FUNCTION "Line.FCMain" : VOID	// FC 50
VERSION : 0.1
VAR_TEMP
  Alarm_Emergency : BOOL ;
  Rich_manuale : BOOL ;
  Rich_automatico : BOOL ;
END_VAR
BEGIN
NETWORK
TITLE =
      CALL  "Line.FCMapE";
      CALL  "Line.FCConfig";
NETWORK
TITLE =
      CALL  "Bench.Alarms" (
           NumDBallarmi             := "Line.Alarms",
           Reset_Allarmi            := "Line.Systems".Command.Reset_allarmi,
           AllarmeEmergenza         := "Line".Diagnostic.Alarm_Emergency,
           AllarmeStopCiclo         := "Line".Diagnostic.Alarm_Stop_Cycle,
           AllarmeStartCiclo        := "Line".Diagnostic.Alarm_No_Restart,
           AllarmeWarning           := "Line".Diagnostic.Alarm_Warning);
// cumula gli stati di emergenza per evitare definizioni errate degli stati macchina!
      A     "Line".Diagnostic.Alarm_Emergency;
      O     "OP10".Diagnostic.Alarm_Emergency;
      O     "OP20".Diagnostic.Alarm_Emergency;
      O     "OP40".Diagnostic.Alarm_Emergency;
      =     #Alarm_Emergency;
      A     "Line.MapE".S_Manuale;
      =     #Rich_manuale;
      A     "Line.MapE".S_Automatico;
      A     "Line.Systems".State.Porte_chiuse;
      =     #Rich_automatico;
      CALL  "Bench.Mode" (
           Enable                   := TRUE,
           AllarmeEmergenza         := #Alarm_Emergency,
           AusiliariOK              := "Line.MapE".Aux_OK,
           ComandoTestMacchina      := FALSE,
           ComandoSetup             := FALSE,
           ComandoManuale           := #Rich_manuale,
           ComandoAutomatico        := #Rich_automatico,
           TimerTest                := T 1,
           ModoEmergenza            := "Line".Mode.Emergency,
           ModoTestMacchina         := "Line".Mode.Test_Machine,
           ModoSetup                := "Line".Mode.Setup,
           ModoManuale              := "Line".Mode.Manual,
           ModoAutomatico           := "Line".Mode.Automatic,
           DO_PlcOk                 := "Line.Systems".State.PLC_OK);
      A     "Line.MapE".S_Manuale;
      FP    "M100.3";
      =     "FP_manual";
      A     "Line.MapE".S_Automatico;
      FP    "M100.5";
      =     "Fp_Automatic";
      A     "FP_manual";
      O     "Fp_Automatic";
      ON    "Line.MapE".Aux_OK;
      R     "Line.OperatorPanel".States.Op10_recipe;
      R     "Line.OperatorPanel".States.Op20_recipe;
      R     "Line.OperatorPanel".States.Op40_recipe;
NETWORK
TITLE =
      CALL  "Line.FCSystems";
      CALL  "Line.FCOperatorPanel";
      CALL  "Line.FCCycles";
NETWORK
TITLE =
      CALL  "Line.FCMapA";
END_FUNCTION

FUNCTION "Line.FCMapE" : VOID	// FC 51
VERSION : 0.1
BEGIN
NETWORK
TITLE =
      A     I 0.0;
      =     "Line.MapE".Q_Ribaditrice;
      A     I 0.1;
      =     "Line.MapE".Q_protezione_uscite;
      A     I 0.2;
      =     "Line.MapE".Q_Protez_circ_emergena;
      A     I 0.3;
      =     "Line.MapE".Q_Automatici_230_V;
      A     I 0.4;
      =     "Line.MapE".Aux_OK;
      A     I 0.5;
      =     "Line.MapE".Ripari_OK;
      A     I 0.6;
      =     "Line.MapE".Anomalia_Condizionatore;
      A     I 0.7;
      =     "Line.MapE".Sequenza_fasi_OK;
NETWORK
TITLE =
      A     I 1.0;
      =     "Line.MapE".PLC_OK;
      A     I 1.1;
      =     "Line.MapE".Chiave_Blocc_Porta_SX;
      A     I 1.2;
      =     "Line.MapE".Chiave_Blocc_Porta_DX;
      A     I 1.3;
      =     "Line.MapE".P_TestLampade;
      A     I 1.4;
      =     "Line.MapE".P_StartCiclo;
      AN    I 1.5;
      =     "Line.MapE".P_StopCiclo;
      A     I 1.7;
      =     "Line.MapE".S_Manuale;
      A     I 1.6;
      =     "Line.MapE".S_Automatico;
NETWORK
TITLE =
      A     I 2.0;
      =     "Line.MapE".Q_Azionam_Asse_X;
      A     I 2.1;
      =     "Line.MapE".Q_Azionam_Asse_Y;
      A     I 6.2;
      =     "Line.MapE".Jog_piu;
      A     I 6.3;
      =     "Line.MapE".Jog_meno;
      A     I 6.4;
      =     "Line.MapE".P_reset_allarmi;
      A     I 6.5;
      =     "Line.MapE".Pressostato_aria;
      A     I 7.6;
      =     "Line.MapE".Ribaditrice_bassa;
      A     I 7.5;
      =     "Line.MapE".Ribaditrice_alta;
NETWORK
TITLE =
      A     I 6.6;
      =     "Line.MapE".Press_aria_dpoop_EMG;
      A     I 2.2;
      =     "Line.MapE".Extracorsa_X;
      A     I 4.7;
      =     "Line.MapE".Extracorsa_Y;
END_FUNCTION

FUNCTION "Line.FCMapA" : VOID	// FC 52
VERSION : 0.1
BEGIN
NETWORK
TITLE =
      A     "Line.MapA".PLC_OK;
      =     Q 0.0;
// tolto!
//      UN    "Line.MapA".Valvola_generale_aria
//      =     A      3.5
      A     "Line.MapA".Marcia_ribaditrice;
      =     Q 1.0;
      A     "Line.MapA".EV_abbassa_ribaditrice;
      =     Q 1.1;
//      U     "Line.MapA".Spare_0_4
//      =     A      1.2
      A     "Line.MapA".Blocco_porta_SX;
      =     Q 3.6;
      A     "Line.MapA".Blocco_porta_DX;
      =     Q 3.7;
      A     "Line.MapA".Lampeggiante_allarmi;
      =     Q 0.7;
      A     "Line.MapA".LampPorteChiuse;
      =     Q 1.7;
END_FUNCTION

FUNCTION "Line.FCConfig" : VOID	// FC 53
VERSION : 0.1
BEGIN
NETWORK
TITLE =
      L     L#100;
      T     "Line.Config".Accel_assi_auto;
      T     "Line.Config".Accel_assi_man;
// Impostate da pagina Config su OP
//      L     L#15000
//      T     "Line.Config".Vel_max_assi_auto
////      T     "Line.Config".Vel_max_assi_man
//      L     L#71501
//      T     "Line.Config".Offset_attrezzo_OP10_X
//      L     L#47116
//      T     "Line.Config".Offset_attrezzo_OP10_Y
//      L     L#371523
//      T     "Line.Config".Offset_attrezzo_OP40_X
//      L     L#47047
//      T     "Line.Config".Offset_attrezzo_OP40_Y
END_FUNCTION

FUNCTION "Line.FCSystems" : VOID	// FC 55
VERSION : 0.1
VAR_TEMP
  Cmd_Marcia_ribaditrice : BOOL ;
  Cmd_Marcia_ribaditr_ibl : BOOL ;
  Cmd_abbassa_rib : BOOL ;
  Cmd_alza_rib : BOOL ;
  Cmd_abbassa_rib_ibl : BOOL ;
  Cmd_alza_rib_ibl : BOOL ;
  StartPosizX : BOOL ;
  StartPosizX_ibl : BOOL ;
  JogPiuX : BOOL ;
  JogMenoX : BOOL ;
  JogPiuX_ibl : BOOL ;
  JogMenoX_ibl : BOOL ;
  StartPosizY : BOOL ;
  StartPosizY_ibl : BOOL ;
  JogPiuY : BOOL ;
  JogMenoY : BOOL ;
  JogPiuY_ibl : BOOL ;
  JogMenoY_ibl : BOOL ;
  Profi_w_error : BOOL ;
  Profi_r_error : BOOL ;
  Override : INT ;
  Velocita_asse_X : DINT ;
  Velocita_asse_Y : DINT ;
  TeachIn_page_OP10 : BOOL ;
  TeachIn_page_OP40 : BOOL ;
  Punt1 : DINT ;
  PuntoSelezionato : INT ;
  Pos_comandata_asse_X : DINT ;
  Pos_comandata_asse_Y : DINT ;
  Tempo_ribaditura : DINT ;
END_VAR
BEGIN
NETWORK
TITLE = ******************       Diagnostica       *******************
NETWORK
TITLE = Diagnostica: Reset Allarmi
      A     "Line.MapE".P_reset_allarmi;
      FP    "AppoFP_M50.0";
      O(;
      A     "Line.OperatorPanel".Commands.Reset_Allarmi;
      FP    "AppoFP_M50.1";
      );
      S     "Line.Systems".Command.Reset_allarmi;
      A     "Line.Systems".Command.Reset_allarmi;
      L     S5T#500MS;
      SD    "TempoResetAllarmi";
      A     "TempoResetAllarmi";
      R     "Line.Systems".Command.Reset_allarmi;
NETWORK
TITLE = Allarmi di emergenza
      AN    "Line.MapE".Q_protezione_uscite;
      O(;
      A     "Line.Alarms".Emegency.Alarm01;
      AN    "Line.Systems".Command.Reset_allarmi;
      );
      =     "Line.Alarms".Emegency.Alarm01;
      AN    "Line.MapE".Q_Protez_circ_emergena;
      O(;
      A     "Line.Alarms".Emegency.Alarm02;
      AN    "Line.Systems".Command.Reset_allarmi;
      );
      =     "Line.Alarms".Emegency.Alarm02;
      AN    "Line.MapE".Sequenza_fasi_OK;
      =     "Line.Alarms".Emegency.Alarm03;
      AN    "Line.MapE".Q_Azionam_Asse_X;
      O(;
      A     "Line.Alarms".Emegency.Alarm04;
      AN    "Line.Systems".Command.Reset_allarmi;
      );
      =     "Line.Alarms".Emegency.Alarm04;
      AN    "Line.MapE".Q_Azionam_Asse_Y;
      O(;
      A     "Line.Alarms".Emegency.Alarm05;
      AN    "Line.Systems".Command.Reset_allarmi;
      );
      =     "Line.Alarms".Emegency.Alarm05;
      A     "Line.MapA".PLC_OK;
      AN    "Line.MapE".PLC_OK;
      O(;
      AN    "Line.MapA".PLC_OK;
      A     "Line.MapE".PLC_OK;
      );
      L     S5T#500MS;
      SD    "T_All_Rientro_PLC_OK";
      A     "T_All_Rientro_PLC_OK";
      S     "Line.Alarms".Emegency.Alarm14;
NETWORK
TITLE = Extracorsa Assi: Allarmi Emergenza
NETWORK
TITLE = Allarmi di STOP CICLO
      AN    "Line.MapE".Aux_OK;
      =     "Line.Alarms".StopCycle.Alarm11;
NETWORK
TITLE = Allarmi di NON START CICLO
NETWORK
TITLE = Allarmi di Warning
      AN    "Line.MapE".Q_Ribaditrice;
//      O(    
//      U     DB54.DBX   24.0
//      UN    DB55.DBX    0.0
//      )     
      =     "Line.Alarms".Warning.Alarm01;
      AN    "Line.MapE".Q_Automatici_230_V;
      =     "Line.Alarms".Warning.Alarm02;
      A     "Line.MapE".Anomalia_Condizionatore;
      =     "Line.Alarms".Warning.Alarm03;
NETWORK
TITLE = Diagnostica: Hold Macchina
      AN    "Line".Diagnostic.Alarm_Emergency;
      A(;
      A     "Line".Mode.Automatic;
      AN    "Line".Diagnostic.Alarm_Stop_Cycle;
      A     "Line.Systems".State.Porte_chiuse_e_bloccate;
      O(;
      A     "Line".Mode.Manual;
      A     "Line.Systems".State.Porte_chiuse;
      );
      );
      =     "Line".Diagnostic.Safe_State;
NETWORK
TITLE = ******************          Stati            *******************
      A     "Op10.Bench.Systems".State.Cassetto_fuori;
      O     "Op10.Bench.Systems".State.Cassetto_dentro;
      A     "Op10.Bench.Systems".State.Index_cassetto_alto;
      =     "Line.Systems".State.Cassetto_OP10_indexato;
      A     "Op40.Bench.Systems".State.Cassetto_fuori;
      O     "Op40.Bench.Systems".State.Cassetto_dentro;
      A     "Op40.Bench.Systems".State.Index_cassetto_alto;
      =     "Line.Systems".State.Cassetto_OP40_indexato;
NETWORK
TITLE =
      A     "Line.MapE".Ripari_OK;
      =     "Line.Systems".State.Porte_chiuse;
NETWORK
TITLE = Stato: Fronte Start Ciclo
NETWORK
TITLE = Lampade
      AN    "Line.Systems".State.Porte_chiuse;
      A     "Clock-T=0,8 sec.";
      O     "Line.Systems".State.Porte_chiuse;
      =     "Line.MapA".LampPorteChiuse;
NETWORK
TITLE = Pagina attiva di TeachIn
// Trovo quale stazione è in pagina di gestione punti
      L     "Line.OperatorPanel".OP_System_Data.PageDisplayed;
      L     21;
      ==I;
      =     #TeachIn_page_OP10;
      L     "Line.OperatorPanel".OP_System_Data.PageDisplayed;
      L     31;
      ==I;
      =     #TeachIn_page_OP40;
NETWORK
TITLE = ******************         Sistemi           *******************
NETWORK
TITLE = Uscita PLC OK
      A     "Line.Systems".State.PLC_OK;
      =     "Line.MapA".PLC_OK;
NETWORK
TITLE = Valvola generale aria
//      UN    "Line".Mode.Emergency
//      =     "Line.MapA".Valvola_generale_aria
      A     "Line.MapE".Aux_OK;
      AN    "Line.MapE".Press_aria_dpoop_EMG;
      O(;
      AN    "Line.MapE".Aux_OK;
      A     "Line.MapE".Press_aria_dpoop_EMG;
      );
      L     S5T#3S;
      SD    "T_Allarme_aria_compressa";
      A     "T_Allarme_aria_compressa";
      A     "Line.MapE".Aux_OK;
      ON    "Line.MapE".Pressostato_aria;
      O(;
      A     "Line.Alarms".Emegency.Alarm06;
      AN    "Line.Systems".Command.Reset_allarmi;
      );
      =     "Line.Alarms".Emegency.Alarm06;
      A     "T_Allarme_aria_compressa";
      AN    "Line.MapE".Aux_OK;
      O(;
      A     "Line.Alarms".Emegency.Alarm07;
      AN    "Line.Systems".Command.Reset_allarmi;
      );
      =     "Line.Alarms".Emegency.Alarm07;
NETWORK
TITLE = Prenotazione ribaditrice
      A     "Op10.Bench.Systems".Command.Prenota_ribaditrice;
      =     "Line.Systems".Command.PrenotaRib_OP10;
      A     "Op40.Bench.Systems".Command.Prenota_ribaditrice;
      =     "Line.Systems".Command.PrenotaRib_OP40;
      A     "Line.Cycles".Coord_Ribaditrice.State.State_Bit[10];
      =     "Line.Systems".State.Ribad_prenotata_da_OP10;
      A     "Line.Cycles".Coord_Ribaditrice.State.State_Bit[20];
      =     "Line.Systems".State.Ribad_prenotata_da_OP40;
NETWORK
TITLE = Marcia ribaditrice
//*************************** COMANDI DA CICLI *************************
      A     "Op10.Bench.Systems".Command.Marcia_ribaditrice;
      A     "Line.Systems".Command.PrenotaRib_OP10;
      O(;
      A     "Op40.Bench.Systems".Command.Marcia_ribaditrice;
      A     "Line.Systems".Command.PrenotaRib_OP40;
      );
      =     "Line.Systems".Command.Marcia_ribaditrice;
//*************************** COMANDI SENZA INTERBLOCCHI ***************
// Autoritenuta comando di marcia manuale
      A     "Line.OperatorPanel".Commands.Man_Marcia_Ribaditrice;
      A     "Line.MapE".Jog_piu;
      O     "Line.Systems".State.Ribadit_Motore_in_marcia;
      A     "Line".Mode.Manual;
      A(;
      AN    "Line.MapE".Jog_meno;
      ON    "Line.OperatorPanel".Commands.Man_Marcia_Ribaditrice;
      );
      AN    "Line.Alarms".Warning.Alarm05;
      A(;
      L     "Line.OperatorPanel".OP_System_Data.PageDisplayed;
      L     20;
      ==I;
      O(;
      L     "Line.OperatorPanel".OP_System_Data.PageDisplayed;
      L     30;
      ==I;
      );
      );
      =     "Line.Systems".Command.Marcia_manuale_ribaditr;
//CMD---------->Comando Marcia ribaditrice
//MANUALE
      A     "Line.Systems".Command.Marcia_manuale_ribaditr;
      A     "Line".Mode.Manual;
//AUTOMATICO
      O(;
      A     "Line".Mode.Automatic;
      AN    "Line".Diagnostic.Hold_State;
      A     "Line.Systems".Command.Marcia_ribaditrice;
      );
//SICUREZZA
      A     "Line".Diagnostic.Safe_State;
      A     "Line.MapE".Q_Ribaditrice;
      =     #Cmd_Marcia_ribaditrice;
//************************** INTERBLOCCHI (E SEGNALAZIONE) ****************************
//MSG---> Segnalazione interblocco Movimento ribaditrice non ammesso con motore ribaditrice in marcia
//      U     "Line.Systems".Command.Reset_allarmi
//      O(    
//      U     "Line.Systems".State.Cassetto_OP10_indexato
//      U     "Line.Systems".State.Cassetto_OP40_indexato
//      )     
//      R     "Line.Alarms".Warning.Alarm05
//      U     #Cmd_Marcia_ribaditrice
//      U(    
//      UN    "Line.Systems".State.Cassetto_OP10_indexato
//      ON    "Line.Systems".State.Cassetto_OP40_indexato
//      )     
//      S     "Line.Alarms".Warning.Alarm05
//************************** COMANDI CON INTERBLOCCHI ******************************
//CMD-------------> Comando Marcia
      A     #Cmd_Marcia_ribaditrice;
      AN    "Line.Alarms".Warning.Alarm05;
      =     #Cmd_Marcia_ribaditr_ibl;
      =     "Line.Systems".State.Ribadit_Motore_in_marcia;
      =     "Line.MapA".Marcia_ribaditrice;
NETWORK
TITLE = Alza/abbassa ribaditrice
//*************************** COMANDI DA CICLI *************************
      A     "Op10.Bench.Systems".Command.Abbassa_ribaditrice;
      A     "Line.Systems".Command.PrenotaRib_OP10;
      O(;
      A     "Op40.Bench.Systems".Command.Abbassa_ribaditrice;
      A     "Line.Systems".Command.PrenotaRib_OP40;
      );
      =     "Line.Systems".Command.Abbassa_ribaditrice;
      A     "Op10.Bench.Systems".Command.Alza_ribaditrice;
      A     "Line.Systems".Command.PrenotaRib_OP10;
      O(;
      A     "Op40.Bench.Systems".Command.Alza_ribaditrice;
      A     "Line.Systems".Command.PrenotaRib_OP40;
      );
      =     "Line.Systems".Command.Alza_ribaditrice;
//*************************** COMANDI SENZA INTERBLOCCHI ***************
//CMD---------->Comando abbassa ribaditrice
//MANUALE
      A     "Line.OperatorPanel".Commands.Man_Alza_Abb_Ribaditrice;
      A     "Line.MapE".Jog_piu;
      A     "Line".Mode.Manual;
//AUTOMATICO
      O(;
      A     "Line".Mode.Automatic;
      AN    "Line".Diagnostic.Hold_State;
      A     "Line.Systems".Command.Abbassa_ribaditrice;
      );
//SICUREZZA
      A     "Line".Diagnostic.Safe_State;
      =     #Cmd_abbassa_rib;
//CMD---------->Comando alza ribaditrice
//MANUALE
      A     "Line.OperatorPanel".Commands.Man_Alza_Abb_Ribaditrice;
      A     "Line.MapE".Jog_meno;
      A     "Line".Mode.Manual;
//AUTOMATICO
      O(;
      A     "Line".Mode.Automatic;
      AN    "Line".Diagnostic.Hold_State;
      A     "Line.Systems".Command.Alza_ribaditrice;
      );
//SICUREZZA
      A     "Line".Diagnostic.Safe_State;
      =     #Cmd_alza_rib;
//************************** INTERBLOCCHI (E SEGNALAZIONE) ****************************
//MSG---> Segnalazione interblocco Movimento ribaditrice non ammesso con motore ribaditrice in marcia
//      U     "Line.Systems".Command.Reset_allarmi
//      O     "Line.Systems".State.Ribadit_Motore_in_marcia
//      R     "Line.Alarms".Warning.Alarm04
//      U     #Cmd_abbassa_rib
//      O     #Cmd_alza_rib
//      Un    "Line.Systems".State.Ribadit_Motore_in_marcia
//      S     "Line.Alarms".Warning.Alarm04
      A     "Line.Systems".Command.Reset_allarmi;
      O(;
      A     "Line.Systems".State.Cassetto_OP10_indexato;
      A     "Line.Systems".State.Cassetto_OP40_indexato;
      );
      R     "Line.Alarms".Warning.Alarm06;
      A     #Cmd_abbassa_rib;
      A(;
      AN    "Line.Systems".State.Cassetto_OP10_indexato;
      ON    "Line.Systems".State.Cassetto_OP40_indexato;
      );
      S     "Line.Alarms".Warning.Alarm06;
//************************** COMANDI CON INTERBLOCCHI ******************************
//CMD-------------> Comando Mensola Contropunta SX
      AN    "Line.Alarms".Warning.Alarm04;
      AN    "Line.Alarms".Warning.Alarm06;
      A     #Cmd_abbassa_rib;
      =     #Cmd_abbassa_rib_ibl;
      AN    "Line.Alarms".Warning.Alarm04;
      A     #Cmd_alza_rib;
      =     #Cmd_alza_rib_ibl;
      CALL  "Std System.Cylinder" , DB 400 (
           IN_Enable                := TRUE,
           IN_Command_CylForward    := #Cmd_abbassa_rib_ibl,
           IN_Command_CylBack       := #Cmd_alza_rib_ibl,
           IN_EndStroke_Forward     := "Line.MapE".Ribaditrice_bassa,
           IN_EndStroke_Back        := "Line.MapE".Ribaditrice_alta,
           IN_Alarms_Reset          := "Line.Systems".Command.Reset_allarmi,
           IN_Alarms_TimeOut        := T#4S,
           IN_Hold_Condition        := FALSE,
           OUT_EV_Forward           := "Line.MapA".EV_abbassa_ribaditrice,
           OUT_State_CylForward     := "Line.Systems".State.Ribaditrice_bassa,
           OUT_State_CylBack        := "Line.Systems".State.Ribaditrice_alta,
           OUT_Alarm_ES_Forward     := "Line.Alarms".StopCycle.Alarm01,
           OUT_Alarm_ES_Back        := "Line.Alarms".StopCycle.Alarm02,
           OUT_Alarm_ForwBack       := "Line.Alarms".StopCycle.Alarm03);
NETWORK
TITLE = Blocco porte
//************************************* COMANDI ***************************************
      A     "Line".Mode.Automatic;
      A     "Line.Systems".State.Porte_chiuse;
      =     "Line.MapA".Blocco_porta_SX;
      =     "Line.MapA".Blocco_porta_DX;
//************************** INTERBLOCCHI (E SEGNALAZIONE) ****************************
// Allamre porte non chiuse
      A     "Line.Systems".Command.Reset_allarmi;
      O     "Line".Mode.Manual;
      R     "Line.Alarms".StopCycle.Alarm04;
      A     "Line".Mode.Automatic;
      AN    "Line.Systems".State.Porte_chiuse;
      S     "Line.Alarms".StopCycle.Alarm04;
// Allarme porte non bloccate
      A     "Line.Systems".Command.Reset_allarmi;
      O     "Line".Mode.Manual;
      R     "Line.Alarms".StopCycle.Alarm05;
      R     "Line.Alarms".StopCycle.Alarm06;
      A     "Line.MapA".Blocco_porta_SX;
      O     "Line.MapA".Blocco_porta_DX;
      L     S5T#1S;
      SD    "Rit_all_potre_non_blocc";
      A     "Rit_all_potre_non_blocc";
      AN    "Line.MapE".Chiave_Blocc_Porta_SX;
      S     "Line.Alarms".StopCycle.Alarm05;
      A     "Rit_all_potre_non_blocc";
      AN    "Line.MapE".Chiave_Blocc_Porta_DX;
      S     "Line.Alarms".StopCycle.Alarm06;
//************************************* STATI ***************************************
      A     "Line.MapA".Blocco_porta_SX;
      A     "Line.MapA".Blocco_porta_DX;
      AN    "Line.Alarms".StopCycle.Alarm04;
      AN    "Line.Alarms".StopCycle.Alarm05;
      AN    "Line.Alarms".StopCycle.Alarm06;
      =     "Line.Systems".State.Porte_chiuse_e_bloccate;
NETWORK
TITLE = Input asse X
      CALL  "Std.Sinamics_Cu_S" , "Ist_CU_asseX" (
           IN_Enable                := TRUE,
           IN_Addr_Read             := W#16#190,
           IN_Addr_Write            := W#16#190,
           OUT_HW_DI1               := "Line.Systems".State.AsseX_ExtracorsaOK,
           OUT_Profibus_Write_Error := #Profi_w_error,
           OUT_Profibus_Read_Error  := #Profi_r_error);	// indirizzo 400
      A     #Profi_w_error;
      O     #Profi_r_error;
      S     "Line.Alarms".Emegency.Alarm10;
      AN    "Line.Systems".State.AsseX_ExtracorsaOK;
      O     "Line.MapE".Extracorsa_X;
      AN    #Profi_w_error;
      AN    #Profi_r_error;
      S     "Line.Alarms".Emegency.Alarm12;
NETWORK
TITLE = Input asse Y
      CALL  "Std.Sinamics_Cu_S" , "Ist_CU_asseY" (
           IN_Enable                := TRUE,
           IN_Addr_Read             := W#16#1AE,
           IN_Addr_Write            := W#16#1AE,
           OUT_HW_DI1               := "Line.Systems".State.AsseY_ExtracorsaOK,
           OUT_Profibus_Write_Error := #Profi_w_error,
           OUT_Profibus_Read_Error  := #Profi_r_error);	// indirizzo 430
      A     #Profi_w_error;
      O     #Profi_r_error;
      S     "Line.Alarms".Emegency.Alarm11;
      AN    "Line.Systems".State.AsseY_ExtracorsaOK;
      O     "Line.MapE".Extracorsa_Y;
      AN    #Profi_w_error;
      AN    #Profi_r_error;
      S     "Line.Alarms".Emegency.Alarm13;
NETWORK
TITLE = Asse X
//*************************** COMANDI DA CICLI *************************
      AN    "Line.Systems".Command.Reset_allarmi;
      O     "Line.Systems".State.AsseX_Pronto;
      A     "Line".Diagnostic.Safe_State;
      A     "Line.Systems".State.AsseX_ExtracorsaOK;
      AN    "Line.MapE".Extracorsa_X;
      =     "Line.Systems".Command.AsseX_Enable;
      A     "Op10.Bench.Systems".Command.Vai_in_posizione_assi;
      A     "Line.Systems".State.Ribad_prenotata_da_OP10;
      O(;
      A     "Op40.Bench.Systems".Command.Vai_in_posizione_assi;
      A     "Line.Systems".State.Ribad_prenotata_da_OP40;
      );
      A     "Line.Systems".State.AsseX_ExtracorsaOK;
      A     "Line.Systems".Command.AsseX_Enable;
      A     "Line.Systems".State.AsseX_Pronto;
      =     "Line.Systems".Command.AsseX_StartPosizionam;
//*************************** COMANDI SENZA INTERBLOCCHI ***************
//CMD---------->Comando posiziona
//MANUALE
      A     #TeachIn_page_OP10;
      O     #TeachIn_page_OP40;
      A     "Line.OperatorPanel".Commands.Cmd_VaiAlPunto;
      A     "Line".Mode.Manual;
//AUTOMATICO
      O(;
      A     "Line".Mode.Automatic;
      AN    "Line".Diagnostic.Hold_State;
      A     "Line.Systems".Command.AsseX_StartPosizionam;
      );
//SICUREZZA
      A     "Line".Diagnostic.Safe_State;
      =     #StartPosizX;
//CMD---------->Comando Jog +
//MANUALE
      A     "Line.OperatorPanel".Commands.Man_Jog_AsseX;
      A     "Line.MapE".Jog_piu;
      A     "Line".Mode.Manual;
//AUTOMATICO
//SICUREZZA
      A     "Line".Diagnostic.Safe_State;
      =     #JogPiuX;
//CMD---------->Comando Jog -
//MANUALE
      A     "Line.OperatorPanel".Commands.Man_Jog_AsseX;
      A     "Line.MapE".Jog_meno;
      A     "Line".Mode.Manual;
//AUTOMATICO
//SICUREZZA
      A     "Line".Diagnostic.Safe_State;
      =     #JogMenoX;
//************************** INTERBLOCCHI (E SEGNALAZIONE) ****************************
//MSG---> Segnalazione interblocco
      A     "Line.Systems".Command.Reset_allarmi;
      O     "Line.Systems".State.Ribaditrice_alta;
      R     "Line.Alarms".StopCycle.Alarm07;
      A     #StartPosizX;
      O     #JogPiuX;
      O     #JogMenoX;
      AN    "Line.Systems".State.Ribaditrice_alta;
      S     "Line.Alarms".StopCycle.Alarm07;
      A     "Line.Systems".Command.Reset_allarmi;
      O(;
      A     "Line.Systems".State.Cassetto_OP10_indexato;
      A     "Line.Systems".State.Cassetto_OP40_indexato;
      );
      R     "Line.Alarms".Warning.Alarm07;
      A     #StartPosizX;
      O     #JogPiuX;
      O     #JogMenoX;
      A(;
      AN    "Line.Systems".State.Cassetto_OP10_indexato;
      ON    "Line.Systems".State.Cassetto_OP40_indexato;
      );
      S     "Line.Alarms".Warning.Alarm07;
//************************** COMANDI CON INTERBLOCCHI ******************************
      AN    "Line.Alarms".StopCycle.Alarm07;
      AN    "Line.Alarms".Warning.Alarm07;
      A     #StartPosizX;
      =     #StartPosizX_ibl;
      AN    "Line.Alarms".StopCycle.Alarm07;
      AN    "Line.Alarms".Warning.Alarm07;
      A     #JogPiuX;
      =     #JogPiuX_ibl;
      AN    "Line.Alarms".StopCycle.Alarm07;
      AN    "Line.Alarms".Warning.Alarm07;
      A     #JogMenoX;
      =     #JogMenoX_ibl;
//*********************************  OVERRIDE  *************************************
      L     "Line.OperatorPanel".Data.Cmd_Override_man;
      A     "Line".Mode.Manual;
      JC    Ovx;
      L     "Line.OperatorPanel".Data.Cmd_Override_auto;
      A     "Line".Mode.Automatic;
      JC    Ovx;
      L     0;
Ovx:  T     #Override;
//*********************************  POSIZIONE  *************************************
      A     "Line.Systems".State.Ribad_prenotata_da_OP10;
      A     "Op10.Bench.Systems".Command.Vai_in_posizione_assi;
      A     "Line".Mode.Automatic;
      JCN   nX10;
      L     "Op10.Bench.Systems".Data.Pos_comandata_asse_X;
      L     "Line.Config".Offset_attrezzo_OP10_X;
      +D;
      T     "Line.Systems".Data.AsseX_PosizioneComandata;
      JU    EnX;
nX10: A     "Line.Systems".State.Ribad_prenotata_da_OP40;
      A     "Op40.Bench.Systems".Command.Vai_in_posizione_assi;
      A     "Line".Mode.Automatic;
      JCN   nX40;
      L     "Op40.Bench.Systems".Data.Pos_comandata_asse_X;
      L     "Line.Config".Offset_attrezzo_OP40_X;
      +D;
      T     "Line.Systems".Data.AsseX_PosizioneComandata;
      JU    EnX;
nX40: A     #TeachIn_page_OP10;
      A     "Line.OperatorPanel".Commands.Cmd_VaiAlPunto;
      A     "Line".Mode.Manual;
      JCN   nXv1;
      L     "Line.OperatorPanel".Data.X_PosPuntoSelezionato;
      L     "Line.Config".Offset_attrezzo_OP10_X;
      +D;
      T     "Line.Systems".Data.AsseX_PosizioneComandata;
      JU    EnX;
nXv1: A     #TeachIn_page_OP40;
      A     "Line.OperatorPanel".Commands.Cmd_VaiAlPunto;
      A     "Line".Mode.Manual;
      JCN   nXv4;
      L     "Line.OperatorPanel".Data.X_PosPuntoSelezionato;
      L     "Line.Config".Offset_attrezzo_OP40_X;
      +D;
      T     "Line.Systems".Data.AsseX_PosizioneComandata;
      JU    EnX;
nXv4: NOP   0;
// Errore di comando posizione
      L     0;
      T     "Line.Systems".Data.AsseX_PosizioneComandata;
EnX:  NOP   0;
//*********************************  VELOCITA'  *************************************
// limita velocità massima di ricetta
      A     "Line.Systems".State.Ribad_prenotata_da_OP40;
      JC    x40;
      L     "Op10.Bench.Recipe".Velocita_asse_X;
      T     #Velocita_asse_X;
      JU    x10;
x40:  L     "Op40.Bench.Recipe".Velocita_asse_X1;
      T     #Velocita_asse_X;
x10:  NOP   0;
      L     #Velocita_asse_X;
      L     "Line.Config".Vel_max_assi_auto;
      <D;
      JC    m1x;
      L     "Line.Config".Vel_max_assi_auto;
      T     #Velocita_asse_X;
m1x:  NOP   0;
// imposta velcità automatico
      A     "Line".Mode.Automatic;
      JCN   nVaX;
      L     #Velocita_asse_X;
      T     "Line.Systems".Data.AsseX_Velocita;
      L     "Line.Config".Accel_assi_auto;
      T     "Line.Systems".Data.AsseX_Accelerazione;
      T     "Line.Systems".Data.AsseX_Decellerazione;
      JU    nVmX;
// imposta velocità manuale
nVaX: L     "Line.Config".Vel_max_assi_man;
      T     "Line.Systems".Data.AsseX_Velocita;
      L     "Line.Config".Accel_assi_man;
      T     "Line.Systems".Data.AsseX_Accelerazione;
      T     "Line.Systems".Data.AsseX_Decellerazione;
nVmX: NOP   0;
      CALL  "Std_Sinamics_Axis" , "Ist_AsseX" (
           Enable_Function          := TRUE,
           AddrIN                   := W#16#194,
           AddrOUT                  := W#16#194,
           Cmd_Jog_Minus_Axis       := #JogMenoX_ibl,
           Cmd_Jog_Plus_Axis        := #JogPiuX_ibl,
           Cmd_Start_Posit_Axis     := #StartPosizX_ibl,
           Cmd_Reference_Axis       := "Dummy_ReferenceAxX",
           In_Reference_Cam         := "Dummy_RefCamAxX",
           Cmd_Enable_Axis          := "Line.Systems".Command.AsseX_Enable,
           Cmd_ResetAlarm           := "Line.Systems".Command.Reset_allarmi,
           Cmd_Override_Axis        := #Override,
           Cmd_Acceleration_Axis    := "Line.Systems".Data.AsseX_Accelerazione,
           Cmd_Deceleration_Axis    := "Line.Systems".Data.AsseX_Decellerazione,
           Cmd_Speed_Axis           := "Line.Systems".Data.AsseX_Velocita,
           Cmd_Position_Axis        := "Line.Systems".Data.AsseX_PosizioneComandata,
           Cmd_Positioning_Mode     := 0,
           Profibus_Write_Error     := #Profi_w_error,
           Profibus_Read_Error      := #Profi_r_error,
           St_Referenced_Axis       := "Line.Systems".State.AsseX_referenziato,
           St_Pos_Axis_OK           := "Line.Systems".State.AsseX_posizioneRaggiunta,
           St_Axis_Running          := "Line.Systems".State.AsseX_inMovimento,
           St_Alarm_Code_Axis       := "Line.Systems".Data.AsseX_CodiceErrore,
           St_Position_Axis         := "Line.Systems".Data.AsseX_PosizioneAttuale,
           St_EndstrokePlus_Reached := "Line.Systems".State.AsseX_FC_avanti,
           St_EndstrokeMinu_Reached := "Line.Systems".State.AsseX_FC_indietro,
           St_Axis_ReadyToStart     := "Line.Systems".State.AsseX_Pronto);	// indirizzo 404
      A     #Profi_w_error;
      O     #Profi_r_error;
      S     "Line.Alarms".Emegency.Alarm08;
NETWORK
TITLE = Asse Y
//*************************** COMANDI DA CICLI *************************
      AN    "Line.Systems".Command.Reset_allarmi;
      O     "Line.Systems".State.AsseY_pronto;
      A     "Line".Diagnostic.Safe_State;
      A     "Line.Systems".State.AsseY_ExtracorsaOK;
      AN    "Line.MapE".Extracorsa_Y;
      =     "Line.Systems".Command.AsseY_Enable;
      A     "Op10.Bench.Systems".Command.Vai_in_posizione_assi;
      A     "Line.Systems".State.Ribad_prenotata_da_OP10;
      O(;
      A     "Op40.Bench.Systems".Command.Vai_in_posizione_assi;
      A     "Line.Systems".State.Ribad_prenotata_da_OP40;
      );
      A     "Line.Systems".State.AsseY_ExtracorsaOK;
      A     "Line.Systems".Command.AsseY_Enable;
      A     "Line.Systems".State.AsseY_pronto;
      =     "Line.Systems".Command.AsseY_StartPosizionam;
//*************************** COMANDI SENZA INTERBLOCCHI ***************
//CMD---------->Comando posiziona
//MANUALE
      A     #TeachIn_page_OP10;
      O     #TeachIn_page_OP40;
      A     "Line.OperatorPanel".Commands.Cmd_VaiAlPunto;
      A     "Line".Mode.Manual;
//AUTOMATICO
      O(;
      A     "Line".Mode.Automatic;
      AN    "Line".Diagnostic.Hold_State;
      A     "Line.Systems".Command.AsseY_StartPosizionam;
      );
//SICUREZZA
      A     "Line".Diagnostic.Safe_State;
      =     #StartPosizY;
//CMD---------->Comando Jog +
//MANUALE
      A     "Line.OperatorPanel".Commands.Man_Jog_AsseY;
      A     "Line.MapE".Jog_piu;
      A     "Line".Mode.Manual;
//AUTOMATICO
//SICUREZZA
      A     "Line".Diagnostic.Safe_State;
      =     #JogPiuY;
//CMD---------->Comando Jog -
//MANUALE
      A     "Line.OperatorPanel".Commands.Man_Jog_AsseY;
      A     "Line.MapE".Jog_meno;
      A     "Line".Mode.Manual;
//AUTOMATICO
//SICUREZZA
      A     "Line".Diagnostic.Safe_State;
      =     #JogMenoY;
//************************** INTERBLOCCHI (E SEGNALAZIONE) ****************************
//MSG---> Segnalazione interblocco
      A     "Line.Systems".Command.Reset_allarmi;
      O     "Line.Systems".State.Ribaditrice_alta;
      R     "Line.Alarms".StopCycle.Alarm08;
      A     #StartPosizY;
      O     #JogPiuY;
      O     #JogMenoY;
      AN    "Line.Systems".State.Ribaditrice_alta;
      S     "Line.Alarms".StopCycle.Alarm08;
// una segnalazione per entrambi gli assi: reset su gestione asse X
      A     #StartPosizY;
      O     #JogPiuY;
      O     #JogMenoY;
      A(;
      AN    "Line.Systems".State.Cassetto_OP10_indexato;
      ON    "Line.Systems".State.Cassetto_OP40_indexato;
      );
      S     "Line.Alarms".Warning.Alarm07;
//************************** COMANDI CON INTERBLOCCHI ******************************
      AN    "Line.Alarms".StopCycle.Alarm08;
      AN    "Line.Alarms".Warning.Alarm07;
      A     #StartPosizY;
      =     #StartPosizY_ibl;
      AN    "Line.Alarms".StopCycle.Alarm08;
      AN    "Line.Alarms".Warning.Alarm07;
      A     #JogPiuY;
      =     #JogPiuY_ibl;
      AN    "Line.Alarms".StopCycle.Alarm08;
      AN    "Line.Alarms".Warning.Alarm07;
      A     #JogMenoY;
      =     #JogMenoY_ibl;
//*********************************  OVERRIDE  *************************************
      L     "Line.OperatorPanel".Data.Cmd_Override_man;
      A     "Line".Mode.Manual;
      JC    Ovy;
      L     "Line.OperatorPanel".Data.Cmd_Override_auto;
      A     "Line".Mode.Automatic;
      JC    Ovy;
      L     0;
Ovy:  T     #Override;
//*********************************  POSIZIONE  *************************************
      A     "Line.Systems".State.Ribad_prenotata_da_OP10;
      A     "Op10.Bench.Systems".Command.Vai_in_posizione_assi;
      A     "Line".Mode.Automatic;
      JCN   nY10;
      L     "Op10.Bench.Systems".Data.Pos_comandata_asse_Y;
      L     "Line.Config".Offset_attrezzo_OP10_Y;
      +D;
      T     "Line.Systems".Data.AsseY_PosizioneComandata;
      JU    EnY;
nY10: A     "Line.Systems".State.Ribad_prenotata_da_OP40;
      A     "Op40.Bench.Systems".Command.Vai_in_posizione_assi;
      A     "Line".Mode.Automatic;
      JCN   nY40;
      L     "Op40.Bench.Systems".Data.Pos_comandata_asse_Y;
      L     "Line.Config".Offset_attrezzo_OP40_Y;
      +D;
      T     "Line.Systems".Data.AsseY_PosizioneComandata;
      JU    EnY;
nY40: A     #TeachIn_page_OP10;
      A     "Line.OperatorPanel".Commands.Cmd_VaiAlPunto;
      A     "Line".Mode.Manual;
      JCN   nYv1;
      L     "Line.OperatorPanel".Data.Y_PosPuntoSelezionato;
      L     "Line.Config".Offset_attrezzo_OP10_Y;
      +D;
      T     "Line.Systems".Data.AsseY_PosizioneComandata;
      JU    EnY;
nYv1: A     #TeachIn_page_OP40;
      A     "Line.OperatorPanel".Commands.Cmd_VaiAlPunto;
      A     "Line".Mode.Manual;
      JCN   nYv4;
      L     "Line.OperatorPanel".Data.Y_PosPuntoSelezionato;
      L     "Line.Config".Offset_attrezzo_OP40_Y;
      +D;
      T     "Line.Systems".Data.AsseY_PosizioneComandata;
      JU    EnY;
nYv4: NOP   0;
// Errore di comando posizione
      L     0;
      T     "Line.Systems".Data.AsseY_PosizioneComandata;
EnY:  NOP   0;
//*********************************  VELOCITA'  *************************************
// limita velocità massima di ricetta
      A     "Line.Systems".State.Ribad_prenotata_da_OP40;
      JC    y40;
      L     "Op10.Bench.Recipe".Velocita_asse_Y;
      T     #Velocita_asse_Y;
      JU    y10;
y40:  L     "Op40.Bench.Recipe".Velocita_asse_Y1;
      T     #Velocita_asse_Y;
y10:  NOP   0;
      L     #Velocita_asse_Y;
      L     "Line.Config".Vel_max_assi_auto;
      <D;
      JC    m1Y;
      L     "Line.Config".Vel_max_assi_auto;
      T     #Velocita_asse_Y;
m1Y:  NOP   0;
// imposta velcità automatico
      A     "Line".Mode.Automatic;
      JCN   nVaY;
      L     #Velocita_asse_Y;
      T     "Line.Systems".Data.AsseY_Velocita;
      L     "Line.Config".Accel_assi_auto;
      T     "Line.Systems".Data.AsseY_Accelerazione;
      T     "Line.Systems".Data.AsseY_Decellerazione;
      JU    nVmY;
// imposta velocità manuale
nVaY: L     "Line.Config".Vel_max_assi_man;
      T     "Line.Systems".Data.AsseY_Velocita;
      L     "Line.Config".Accel_assi_man;
      T     "Line.Systems".Data.AsseY_Accelerazione;
      T     "Line.Systems".Data.AsseY_Decellerazione;
nVmY: NOP   0;
      CALL  "Std_Sinamics_Axis" , "Ist_AsseY" (
           Enable_Function          := TRUE,
           AddrIN                   := W#16#1B2,
           AddrOUT                  := W#16#1B2,
           Cmd_Jog_Minus_Axis       := #JogMenoY_ibl,
           Cmd_Jog_Plus_Axis        := #JogPiuY_ibl,
           Cmd_Start_Posit_Axis     := #StartPosizY_ibl,
           Cmd_Reference_Axis       := "Dummy_ReferenceAxY",
           In_Reference_Cam         := "Dummy_RefCamAxY",
           Cmd_Enable_Axis          := "Line.Systems".Command.AsseY_Enable,
           Cmd_ResetAlarm           := "Line.Systems".Command.Reset_allarmi,
           Cmd_Override_Axis        := #Override,
           Cmd_Acceleration_Axis    := "Line.Systems".Data.AsseY_Accelerazione,
           Cmd_Deceleration_Axis    := "Line.Systems".Data.AsseY_Decellerazione,
           Cmd_Speed_Axis           := "Line.Systems".Data.AsseY_Velocita,
           Cmd_Position_Axis        := "Line.Systems".Data.AsseY_PosizioneComandata,
           Cmd_Positioning_Mode     := 0,
           Profibus_Write_Error     := #Profi_w_error,
           Profibus_Read_Error      := #Profi_r_error,
           St_Referenced_Axis       := "Line.Systems".State.AsseY_referenziato,
           St_Pos_Axis_OK           := "Line.Systems".State.AsseY_posizioneRaggiunta,
           St_Axis_Running          := "Line.Systems".State.AsseY_inMovimento,
           St_Alarm_Code_Axis       := "Line.Systems".Data.AsseY_CodiceErrore,
           St_Position_Axis         := "Line.Systems".Data.AsseY_PosizioneAttuale,
           St_EndstrokePlus_Reached := "Line.Systems".State.AsseY_FC_avanti,
           St_EndstrokeMinu_Reached := "Line.Systems".State.AsseY_FC_indietro,
           St_Axis_ReadyToStart     := "Line.Systems".State.AsseY_pronto);	// indirizzo 434
      A     #Profi_w_error;
      O     #Profi_r_error;
      S     "Line.Alarms".Emegency.Alarm08;
NETWORK
TITLE = Gestioen bit "Vai al punto" da TeachIn page
      AN    "Line.Systems".State.AsseY_inMovimento;
      AN    "Line.Systems".State.AsseX_inMovimento;
      A     "Line.OperatorPanel".Commands.Cmd_VaiAlPunto;
      L     S5T#500MS;
      SD    T 15;
      AN    #TeachIn_page_OP10;
      AN    #TeachIn_page_OP40;
      O     T 15;
      O     "Line.MapE".P_StopCiclo;
      R     "Line.OperatorPanel".Commands.Cmd_VaiAlPunto;
NETWORK
TITLE = Leggi punto TeachIn page
// catturo momento di ingresso in pagina di teachIn
      A     #TeachIn_page_OP10;
      O     #TeachIn_page_OP40;
      FP    "AppoFPM51.2";
      =     "Line.Systems".State.FP_IngressoInPag_TeachIn;
// Modificato numero del punto
      L     "Line.OperatorPanel".Data.Cmd_PuntoSelezionato;
      L     "Line.Systems".Data.PuntoInTeachIn;
      <>I;
      =     "Line.Systems".State.FP_NumPuntoCambiato;
      L     "Line.OperatorPanel".Data.Cmd_PuntoSelezionato;
      T     "Line.Systems".Data.PuntoInTeachIn;
// Richiesta lettura punto da operatore
      A     "Line.OperatorPanel".Commands.Cmd_LeggiPunto;
      FP    "AppoFPM51.3";
      =     "Line.Systems".State.FP_RichiestaLeggiPunto;
      A     "Line.OperatorPanel".Commands.Cmd_LeggiPunto;
      R     "Line.OperatorPanel".Commands.Cmd_LeggiPunto;
// Funzione di lettura dei dati del punto selezionato
      A     "Line.Systems".State.FP_IngressoInPag_TeachIn;
      O     "Line.Systems".State.FP_NumPuntoCambiato;
      O     "Line.Systems".State.FP_RichiestaLeggiPunto;
      JCN   noLP;
// Azzero le variabili
      L     L#0;
      T     "Line.OperatorPanel".Data.X_PosPuntoSelezionato;
      T     "Line.OperatorPanel".Data.Y_PosPuntoSelezionato;
      T     "Line.OperatorPanel".Data.TempoRibad_PuntoSelez;
// controllo di esser in tabella (punto coerente)
      L     "Line.OperatorPanel".Data.Cmd_PuntoSelezionato;
      L     "Line.OperatorPanel".Data.Min_PerSelezionePunto;
      <I;
      O(;
      L     "Line.OperatorPanel".Data.Cmd_PuntoSelezionato;
      L     "Line.OperatorPanel".Data.Max_PerSelezionePunto;
      >I;
      );
      JC    noLP;
// Sceglie tabella in funzione della stazione OP10 o OP40
      L     "Line.OperatorPanel".Data.Cmd_PuntoSelezionato;
      T     #PuntoSelezionato;
      A     #TeachIn_page_OP40;
      JC    op2;
      OPN   "Op10.Bench.Recipe";
      JU    op1;
op2:  OPN   "Op40.Bench.Recipe";
op1:  NOP   0;
// Leggo i dati del punto
      L     #PuntoSelezionato;
      L     1;
      -I;
      ITD;
      L     L#12;
      *D;
      L     L#82;
      +D;
      SLW   3;
      T     #Punt1;
      L     DBD [#Punt1];
      T     #Pos_comandata_asse_X;
      L     #Punt1;
      L     32;
      +D;
      T     #Punt1;
      L     DBD [#Punt1];
      T     #Pos_comandata_asse_Y;
      L     #Punt1;
      L     32;
      +D;
      T     #Punt1;
      L     DBD [#Punt1];
      T     #Tempo_ribaditura;
      L     #Pos_comandata_asse_X;
      T     "Line.OperatorPanel".Data.X_PosPuntoSelezionato;
      L     #Pos_comandata_asse_Y;
      T     "Line.OperatorPanel".Data.Y_PosPuntoSelezionato;
      L     #Tempo_ribaditura;
      T     "Line.OperatorPanel".Data.TempoRibad_PuntoSelez;
noLP: NOP   0;
NETWORK
TITLE = teachIn punto
// Richiesta TeachIn punto da operatore
      A     "Line.OperatorPanel".Commands.Cmd_TeachInPunto;
      FP    "AppoFPM51.5";
      =     "Line.Systems".State.FP_RichiestaTeachInPunto;
      A     "Line.OperatorPanel".Commands.Cmd_TeachInPunto;
      R     "Line.OperatorPanel".Commands.Cmd_TeachInPunto;
// Funzione di TeachIn del punto selezionato
      A     "Line.Systems".State.FP_RichiestaTeachInPunto;
      JCN   noTI;
      AN    #TeachIn_page_OP10;
      JC    NT10;
//OP10
      L     "Line.OperatorPanel".Data.AsseX_PosAttualeOP10;
      T     "Line.OperatorPanel".Data.X_PosPuntoSelezionato;
      L     "Line.OperatorPanel".Data.AsseY_PosAttualeOP10;
      T     "Line.OperatorPanel".Data.Y_PosPuntoSelezionato;
      JU    noTI;
NT10: AN    #TeachIn_page_OP40;
      JC    NT40;
//OP40
      L     "Line.OperatorPanel".Data.AsseX_PosAttualeOP40;
      T     "Line.OperatorPanel".Data.X_PosPuntoSelezionato;
      L     "Line.OperatorPanel".Data.AsseY_PosAttualeOP40;
      T     "Line.OperatorPanel".Data.Y_PosPuntoSelezionato;
NT40: NOP   0;
noTI: NOP   0;
NETWORK
TITLE = Salva punto
// Richiesta scrittura punto da operatore
      A     "Line.OperatorPanel".Commands.Cmd_SalvaPunto;
      FP    "AppoFPM51.4";
      =     "Line.Systems".State.FP_RichiestaSalvaPunto;
      A     "Line.OperatorPanel".Commands.Cmd_SalvaPunto;
      R     "Line.OperatorPanel".Commands.Cmd_SalvaPunto;
// Funzione di lettura dei dati del punto selezionato
      A     "Line.Systems".State.FP_RichiestaSalvaPunto;
      JCN   noSP;
// controllo di esser in tabella (punto coerente)
      L     "Line.OperatorPanel".Data.Cmd_PuntoSelezionato;
      L     "Line.OperatorPanel".Data.Min_PerSelezionePunto;
      <I;
      O(;
      L     "Line.OperatorPanel".Data.Cmd_PuntoSelezionato;
      L     "Line.OperatorPanel".Data.Max_PerSelezionePunto;
      >I;
      );
      JC    noSP;
// Sceglie tabella in funzione della stazione OP10 o OP40
// Salvo i dati del punto
      L     "Line.OperatorPanel".Data.X_PosPuntoSelezionato;
      T     #Pos_comandata_asse_X;
      L     "Line.OperatorPanel".Data.Y_PosPuntoSelezionato;
      T     #Pos_comandata_asse_Y;
      L     "Line.OperatorPanel".Data.TempoRibad_PuntoSelez;
      T     #Tempo_ribaditura;
      L     "Line.OperatorPanel".Data.Cmd_PuntoSelezionato;
      T     #PuntoSelezionato;
      A     #TeachIn_page_OP40;
      JC    opS2;
      OPN   "Op10.Bench.Recipe";
      JU    opS1;
opS2: OPN   "Op40.Bench.Recipe";
opS1: NOP   0;
      L     #PuntoSelezionato;
      L     1;
      -I;
      ITD;
      L     L#12;
      *D;
      L     L#82;
      +D;
      SLW   3;
      T     #Punt1;
      L     #Pos_comandata_asse_X;
      T     DBD [#Punt1];
      L     #Punt1;
      L     32;
      +D;
      T     #Punt1;
      L     #Pos_comandata_asse_Y;
      T     DBD [#Punt1];
      L     #Punt1;
      L     32;
      +D;
      T     #Punt1;
      L     #Tempo_ribaditura;
      T     DBD [#Punt1];
noSP: NOP   0;
END_FUNCTION

FUNCTION "Line.FCCycles" : VOID	// FC 60
VERSION : 0.1
BEGIN
NETWORK
TITLE =
NETWORK
TITLE =
      A     "Line".Mode.Automatic;
      AN    "Line".Diagnostic.Alarm_Stop_Cycle;
      AN    "Line".Diagnostic.Alarm_Emergency;
// condizione di sicurezza
      =     "Line.Cycles".Coord_Ribaditrice.Command.Activate_Cycle;
      CLR;
      =     "Line".Diagnostic.Hold_State;
      CALL  "Line.Cycle.Coord_ribadit" , "Line.Ist.Cycle.Coord_rib" (
           IN_Cm_ON                 := "Line.Cycles".Coord_Ribaditrice.Command.Activate_Cycle,
           IN_HOLD                  := "Line".Diagnostic.Hold_State,
           IN_STEP                  := FALSE,
           OUT_St_CicloInCorso      := "Line.Cycles".Coord_Ribaditrice.State.Cycle_In_Progress,
           OUT_St_CicloTerminatoOK  := "Line.Cycles".Coord_Ribaditrice.State.Cycle_Ended_OK,
           OUT_St_CicloTerminatoKO  := "Line.Cycles".Coord_Ribaditrice.State.Cycle_Ended_KO,
           OUT_CicloStato           := "Line.Cycles".Coord_Ribaditrice.State.State,
           OUT_Page                 := "Line.Cycles".Coord_Ribaditrice.State.Page,
           OUT_Message              := "Line.Cycles".Coord_Ribaditrice.State.Message);
END_FUNCTION

FUNCTION "Line.FCOperatorPanel" : VOID	// FC 70
VERSION : 0.1
VAR_TEMP
  PagManualeVis : BOOL ;
  PagAutomaticoVis : BOOL ;
  PagDiagnosticVis : BOOL ;
  PagFake : BOOL ;
END_VAR
BEGIN
NETWORK
TITLE = Controlla pagina attiva
// Contollo se visualizzata una pagina automatica o manuale
      L     "Line.OperatorPanel".OP_System_Data.PageDisplayed;
      L     90;
      <=I;
      =     #PagManualeVis;
      L     "Line.OperatorPanel".OP_System_Data.PageDisplayed;
      L     149;
      <=I;
      A(;
      L     "Line.OperatorPanel".OP_System_Data.PageDisplayed;
      L     110;
      >=I;
      );
      =     #PagAutomaticoVis;
      L     "Line.OperatorPanel".OP_System_Data.PageDisplayed;
      L     170;
      <=I;
      A(;
      L     "Line.OperatorPanel".OP_System_Data.PageDisplayed;
      L     150;
      >=I;
      );
      =     #PagDiagnosticVis;
      L     "Line.OperatorPanel".OP_System_Data.PageDisplayed;
      L     300;
      ==I;
      =     #PagFake;
NETWORK
TITLE = Forza pagina attva
// Forzo le pagine principali in funzione dello modo abilitato
      A     "Line".Mode.Automatic;
      O     "Line".Mode.Manual;
      A     #PagDiagnosticVis;
      JC    NoF;
      A     #PagManualeVis;
      O     #PagFake;
      A     "Line".Mode.Automatic;
      JC    FAu;
      A     #PagAutomaticoVis;
      O     #PagFake;
      A     "Line".Mode.Manual;
      JC    FMa;
      JU    NoF;
FAu:  L     120;
      T     "Line.OperatorPanel".OP_System_Data.NewPage;
      JU    NoF;
FMa:  L     10;
      T     "Line.OperatorPanel".OP_System_Data.NewPage;
NoF:  NOP   0;
NETWORK
TITLE = Visualizzazione stati sensori
      A     "Line.Systems".State.Ribaditrice_alta;
      =     "Line.OperatorPanel".States.RibaditriceAlta;
      A     "Line.Systems".State.Ribaditrice_bassa;
      =     "Line.OperatorPanel".States.RibaditriceBassa;
      AN    "Line.Systems".State.Ribadit_Motore_in_marcia;
      =     "Line.OperatorPanel".States.RibaditriceFerma;
      A     "Line.Systems".State.Ribadit_Motore_in_marcia;
      =     "Line.OperatorPanel".States.RibaditriceInMarcia;
      A     "Op10.Bench.Systems".State.Index_cassetto_basso;
      =     "Line.OperatorPanel".States.OP10IndexCassSbloccato;
      A     "Op10.Bench.Systems".State.Index_cassetto_alto;
      =     "Line.OperatorPanel".States.OP10IndexCassBloccato;
      A     "Op10.Bench.Systems".State.Pezzo_sbloccato;
      =     "Line.OperatorPanel".States.OP10PezzoSbloccato;
      A     "Op10.Bench.Systems".State.Pezzo_bloccato;
      =     "Line.OperatorPanel".States.OP10PezzoBloccato;
      A     "Line.Systems".State.AsseX_FC_indietro;
      =     "Line.OperatorPanel".States.AsseXIndietro;
      A     "Line.Systems".State.AsseX_FC_avanti;
      =     "Line.OperatorPanel".States.AsseXAvanti;
      A     "Line.Systems".State.AsseY_FC_indietro;
      =     "Line.OperatorPanel".States.AsseYIndietro;
      A     "Line.Systems".State.AsseY_FC_avanti;
      =     "Line.OperatorPanel".States.AsseYAvanti;
      A     "Op20.Bench.Systems".State.Index_cassetto_basso;
      =     "Line.OperatorPanel".States.OP20IndexCassSbloccato;
      A     "Op20.Bench.Systems".State.Index_cassetto_alto;
      =     "Line.OperatorPanel".States.OP20IndexCassBloccato;
      A     "Op20.Bench.Systems".State.Gruppo_piantaggio_alto;
      =     "Line.OperatorPanel".States.OP20GrPiantaggioAlto;
      A     "Op20.Bench.Systems".State.Gruppo_piantaggio_basso;
      =     "Line.OperatorPanel".States.OP20GrPiantaggioBasso;
      A     "Op20.Bench.Systems".State.Piantaggio_alto;
      =     "Line.OperatorPanel".States.OP20PiantaggioAlto;
      A     "Op20.Bench.Systems".State.Piantaggio_basso;
      =     "Line.OperatorPanel".States.OP20PiantaggioBasso;
      A     "Op40.Bench.Systems".State.Index_cassetto_basso;
      =     "Line.OperatorPanel".States.OP40IndexCassSbloccato;
      A     "Op40.Bench.Systems".State.Index_cassetto_alto;
      =     "Line.OperatorPanel".States.OP40IndexCassBloccato;
      A     "Op40.Bench.Systems".State.Pezzo_sbloccato;
      =     "Line.OperatorPanel".States.OP40PezzoSbloccato;
      A     "Op40.Bench.Systems".State.Pezzo_bloccato;
      =     "Line.OperatorPanel".States.OP40PezzoBloccato;
NETWORK
TITLE = Visualizzazione variabili macchina
// Visualizzazione assi
      L     "Line.Systems".Data.AsseX_PosizioneAttuale;
      T     "Line.OperatorPanel".Data.AsseX_PosizioneAttuale;
      L     "Line.Systems".Data.AsseY_PosizioneAttuale;
      T     "Line.OperatorPanel".Data.AsseY_PosizioneAttuale;
// Visualizzazione assi su OP10
      L     "Line.Systems".Data.AsseX_PosizioneAttuale;
      L     "Line.Config".Offset_attrezzo_OP10_X;
      -D;
      T     "Line.OperatorPanel".Data.AsseX_PosAttualeOP10;
      L     "Line.Systems".Data.AsseY_PosizioneAttuale;
      L     "Line.Config".Offset_attrezzo_OP10_Y;
      -D;
      T     "Line.OperatorPanel".Data.AsseY_PosAttualeOP10;
// Visualizzazione assi su OP40
      L     "Line.Systems".Data.AsseX_PosizioneAttuale;
      L     "Line.Config".Offset_attrezzo_OP40_X;
      -D;
      T     "Line.OperatorPanel".Data.AsseX_PosAttualeOP40;
      L     "Line.Systems".Data.AsseY_PosizioneAttuale;
      L     "Line.Config".Offset_attrezzo_OP40_Y;
      -D;
      T     "Line.OperatorPanel".Data.AsseY_PosAttualeOP40;
// Visualizzazione posizione punzone di piantaggio
      L     "Op20.Bench.MapE"._Posizione_Punzone;
      T     "Line.OperatorPanel".Data.PosizionePunzone;
NETWORK
TITLE = Stato macchina
      L     0;
      A     "Line".Mode.Emergency;
      JC    cls;
      L     1;
      A     "Line".Mode.Test_Machine;
      JC    cls;
      L     2;
      A     "Line".Mode.Setup;
      JC    cls;
      L     3;
      A     "Line".Mode.Manual;
      JC    cls;
      L     4;
      A     "Line".Mode.Automatic;
      JC    cls;
      L     0;
cls:  T     "Line.OperatorPanel".cycles.Line_State;
NETWORK
TITLE = Stati cicli
      A     "Op10.Cycles".General.Command.Activate_Cycle;
      =     "Line.OperatorPanel".cycles.OP10_cycle_general;
      A     "Op10.Cycles".Restore.Command.Activate_Cycle;
      =     "Line.OperatorPanel".cycles.OP10_cycle_restore;
      A     "Op20.Cycles".General.Command.Activate_Cycle;
      =     "Line.OperatorPanel".cycles.OP20_cycle_general;
      A     "Op20.Cycles".Restore.Command.Activate_Cycle;
      =     "Line.OperatorPanel".cycles.OP20_cycle_restore;
      A     "Op40.Cycles".General.Command.Activate_Cycle;
      =     "Line.OperatorPanel".cycles.OP40_cycle_general;
      A     "Op40.Cycles".Restore.Command.Activate_Cycle;
      =     "Line.OperatorPanel".cycles.OP40_cycle_restore;
      A     "Op10.Cycles".Restore.Command.Activate_Cycle;
      JC    R10;
      L     "Op10.Cycles".General.State.Message;
      T     "Line.OperatorPanel".cycles.OP10_message;
      JU    M10;
R10:  L     "Op10.Cycles".Restore.State.Message;
      T     "Line.OperatorPanel".cycles.OP10_message;
M10:  NOP   0;
      L     "Op10.Bench.Systems".Data.Num_punto_in_lavorazione;
      T     "Line.OperatorPanel".cycles.OP10_spacer;
      A     "Op20.Cycles".Restore.Command.Activate_Cycle;
      JC    R20;
      L     "Op20.Cycles".General.State.Message;
      T     "Line.OperatorPanel".cycles.OP20_message;
      JU    M20;
R20:  L     "Op20.Cycles".Restore.State.Message;
      T     "Line.OperatorPanel".cycles.OP20_message;
M20:  NOP   0;
      A     "Op40.Cycles".Restore.Command.Activate_Cycle;
      JC    R40;
      L     "Op40.Cycles".General.State.Message;
      T     "Line.OperatorPanel".cycles.OP40_message;
      JU    M40;
R40:  L     "Op40.Cycles".Restore.State.Message;
      T     "Line.OperatorPanel".cycles.OP40_message;
M40:  NOP   0;
      L     "Op40.Bench.Systems".Data.Num_punto_in_lavorazione;
      T     "Line.OperatorPanel".cycles.OP40_spacer;
NETWORK
TITLE = Min / Max punto in teachIn in funzione della ricetta
      L     "Line.OperatorPanel".OP_System_Data.PageDisplayed;
      L     21;
      <>I;
      JC    n10;
      L     1;
      T     "Line.OperatorPanel".Data.Min_PerSelezionePunto;
      L     "Op10.Bench.Recipe".NumeroPosizioni;
      T     "Line.OperatorPanel".Data.Max_PerSelezionePunto;
      JU    n0;
n10:  L     "Line.OperatorPanel".OP_System_Data.PageDisplayed;
      L     31;
      <>I;
      JC    n40;
      L     1;
      T     "Line.OperatorPanel".Data.Min_PerSelezionePunto;
      L     "Op40.Bench.Recipe".NumeroPosizioni;
      T     "Line.OperatorPanel".Data.Max_PerSelezionePunto;
      JU    n0;
n40:  L     1;
      T     "Line.OperatorPanel".Data.Min_PerSelezionePunto;
      T     "Line.OperatorPanel".Data.Max_PerSelezionePunto;
n0:   NOP   0;
END_FUNCTION

FUNCTION "OP10.FCMain" : VOID	// FC 100
VERSION : 0.1
VAR_TEMP
  ErrorToolType : BOOL ;
END_VAR
BEGIN
NETWORK
TITLE =
NETWORK
TITLE = OP10 ToolType error
      CALL  "Op10.Bench.FCMapE";
      CALL  "Op10.Tool.FCMap.E" (
           ToolType                 := "Op10.Bench.Recipe".ToolType,
           ErrorToolType            := #ErrorToolType);
      A     #ErrorToolType;
      AN    "Op10.Bench.Recipe".Disable.CkCodicePortapezzo;
      S     "Op10.Bench.Alarms".StopCycle.Alarm09;
      CALL  "Op10.Bench.FCConfig";
NETWORK
TITLE =
      A     "Line.Systems".Command.Reset_allarmi;
      =     "Op10.Bench.Systems".Command.Reset_allarmi;
      A     "Line.Systems".Command.TestLampade;
      =     "Op10.Bench.Systems".Command.TestLampade;
      A     "Line.Systems".State.Porte_chiuse;
      =     "Op10.Bench.Systems".State.Porte_chiuse;
      A     "Line.Systems".State.Porte_chiuse_e_bloccate;
      =     "Op10.Bench.Systems".State.Porte_chiuse_e_bloccate;
      CALL  "Bench.Alarms" (
           NumDBallarmi             := "Op10.Bench.Alarms",
           Reset_Allarmi            := "Op10.Bench.Systems".Command.Reset_allarmi,
           AllarmeEmergenza         := "OP10".Diagnostic.Alarm_Emergency,
           AllarmeStopCiclo         := "OP10".Diagnostic.Alarm_Stop_Cycle,
           AllarmeStartCiclo        := "OP10".Diagnostic.Alarm_No_Restart,
           AllarmeWarning           := "OP10".Diagnostic.Alarm_Warning);
// Bench mode = Line mode...
      A     "Line".Mode.Emergency;
      =     "OP10".Mode.Emergency;
      A     "Line".Mode.Test_Machine;
      =     "OP10".Mode.Test_Machine;
      A     "Line".Mode.Setup;
      =     "OP10".Mode.Setup;
      A     "Line".Mode.Manual;
      =     "OP10".Mode.Manual;
      A     "Line".Mode.Automatic;
      =     "OP10".Mode.Automatic;
NETWORK
TITLE =
      CALL  "Op10.Bench.FCSystems";
      CALL  "Op10.FCCycles";
//      CALL  "Op10.Operator_Panel"
NETWORK
TITLE =
      CALL  "Op10.Bench.FCMapA";
END_FUNCTION

FUNCTION "Op10.Bench.FCMapE" : VOID	// FC 101
VERSION : 0.1
BEGIN
NETWORK
TITLE = (start ciclo)
      A     I 6.0;
      =     "Op10.Bench.MapE".P_Consenso_operatore;
      AN    I 8.0;
      =     "Op10.Bench.MapE".Cassetto_fuori;
      A     I 8.1;
      =     "Op10.Bench.MapE".Cassetto_dentro;
      A     I 8.3;
      =     "Op10.Bench.MapE".Index_cassetto_Giu;
      A     I 8.2;
      =     "Op10.Bench.MapE".Index_cassetto_Su;
      A     I 8.5;
      =     "Op10.Bench.MapE".Sblocco_pezzo_Giu;
      A     I 8.4;
      =     "Op10.Bench.MapE".Sblocco_pezzo_Su;
      AN    I 1.5;
      =     "Op10.Bench.MapE".PulStopCiclo;
END_FUNCTION

FUNCTION "Op10.Bench.FCMapA" : VOID	// FC 102
VERSION : 0.1
BEGIN
NETWORK
TITLE =
      A     "Op10.Bench.MapA".Fine_ciclo_OK;
      =     Q 0.3;
      A     "Op10.Bench.MapA".Fine_ciclo_NON_OK;
      =     Q 0.4;
      A     "Op10.Bench.MapA".EV_abb_index_cassetto;
      =     Q 2.2;
      A     "Op10.Bench.MapA".EV_alza_index_cassetto;
      =     Q 2.3;
      A     "Op10.Bench.MapA".EV_sblocco_pezzo;
      =     Q 2.5;
      A     "Op10.Bench.MapA".EV_blocco_pezzo;
      =     Q 2.4;
END_FUNCTION

FUNCTION "Op10.Bench.FCConfig" : VOID	// FC 103
VERSION : 0.1
BEGIN
NETWORK
TITLE =
END_FUNCTION

FUNCTION "Op10.Bench.FCSystems" : VOID	// FC 105
VERSION : 0.1
VAR_TEMP
  Cmd_abbassa_indc : BOOL ;
  Cmd_alza_indc : BOOL ;
  Cmd_abbassa_indc_ibl : BOOL ;
  Cmd_alza_indc_ibl : BOOL ;
  Cmd_sblocca_pezzo : BOOL ;
  Cmd_blocca_pezzo : BOOL ;
  Cmd_sblocca_pezzo_ibl : BOOL ;
  Cmd_blocca_pezzo_ibl : BOOL ;
  Punt1 : DINT ;
  TempoTime : TIME ;
  TempoS5T : S5TIME ;
  Pos_comandata_asse_X : DINT ;
  Pos_comandata_asse_Y : DINT ;
  Tempo_ribaditura : DINT ;
END_VAR
BEGIN
NETWORK
TITLE = ******************       Diagnostica       *******************
NETWORK
TITLE = Allarmi di emergenza
NETWORK
TITLE = Controllo toolcode 
      L     DB106.DBB 0;
      L     W#16#1F;
      AW;
      L     "Op10.Bench.Recipe".ToolCode;
      <>I;
      AN    "Op10.Bench.Recipe".Disable.CkCodicePortapezzo;
      S     "Op10.Bench.Alarms".StopCycle.Alarm10;
NETWORK
TITLE = Allarmi di STOP CICLO
NETWORK
TITLE = Controllo anelli adattamento
      A     "Op10.Bench.Recipe".Anello1Abilitato;
      AN    "Op10.Tools.MapE".Anello_1_Inserito;
      O(;
      AN    "Op10.Bench.Recipe".Anello1Abilitato;
      A     "Op10.Tools.MapE".Anello_1_Inserito;
      );
      AN    "Op10.Bench.Recipe".Disable.CkPresAnelloAdattamento;
      S     "Op10.Bench.Alarms".StopCycle.Alarm01;
      A     "Op10.Bench.Recipe".Anello2Abilitato;
      AN    "Op10.Tools.MapE".Anello_2_Inserito;
      O(;
      AN    "Op10.Bench.Recipe".Anello2Abilitato;
      A     "Op10.Tools.MapE".Anello_2_Inserito;
      );
      AN    "Op10.Bench.Recipe".Disable.CkPresAnelloAdattamento;
      S     "Op10.Bench.Alarms".StopCycle.Alarm02;
NETWORK
TITLE = Allarmi di NON START CICLO
NETWORK
TITLE = Allarmi di Warning
NETWORK
TITLE = Diagnostica: Hold Macchina
      AN    "OP10".Diagnostic.Alarm_Emergency;
      A(;
      A     "OP10".Mode.Automatic;
      AN    "OP10".Diagnostic.Alarm_Stop_Cycle;
      A     "Op10.Bench.Systems".State.Porte_chiuse_e_bloccate;
      O(;
      A     "OP10".Mode.Manual;
      A     "Op10.Bench.Systems".State.Porte_chiuse;
      );
      );
      =     "OP10".Diagnostic.Safe_State;
NETWORK
TITLE = ******************          Stati            *******************
      A     "Op10.Bench.MapE".Cassetto_fuori;
      =     "Op10.Bench.Systems".State.Cassetto_fuori;
      A     "Op10.Bench.MapE".Cassetto_dentro;
      =     "Op10.Bench.Systems".State.Cassetto_dentro;
NETWORK
TITLE =
      A     "Line.Systems".State.Ribaditrice_alta;
      =     "Op10.Bench.Systems".State.Ribaditrice_alta;
      A     "Line.Systems".State.Ribaditrice_bassa;
      =     "Op10.Bench.Systems".State.Ribaditrice_bassa;
      A     "Line.Systems".State.Ribadit_Motore_in_marcia;
      =     "Op10.Bench.Systems".State.Ribaditrice_in_marcia;
      AN    "Line.Systems".State.AsseX_inMovimento;
      AN    "Line.Systems".State.AsseY_inMovimento;
      =     "Op10.Bench.Systems".State.Assi_fermi;
NETWORK
TITLE = Stato: Fronte Start Ciclo
      A     "Op10.Bench.MapE".P_Consenso_operatore;
      FP    "AppoFP_M50.2";
      =     "Op10.Bench.Systems".Command.FP_Consenso_operatore;
NETWORK
TITLE = Lampade
      A     "Op10.Bench.Systems".State.Ribaditura_pezzo_OK;
      A     "OP10".Mode.Automatic;
      O     "Op10.Bench.Systems".Command.TestLampade;
      =     "Op10.Bench.MapA".Fine_ciclo_OK;
      A     "Op10.Bench.Systems".State.Ribaditura_pezzo_KO;
      A     "OP10".Mode.Automatic;
      O     "Op10.Bench.Systems".Command.TestLampade;
      =     "Op10.Bench.MapA".Fine_ciclo_NON_OK;
NETWORK
TITLE = Cycle Type
NETWORK
TITLE = ******************         Sistemi           *******************
NETWORK
TITLE = Alza/abbassa Index cassetto
//*************************** COMANDI DA CICLI *************************
      A     "Op10.Cycles".General.State.State_Bit[13];
      O     "Op10.Cycles".General.State.State_Bit[35];
      O     "Op10.Cycles".Restore.State.State_Bit[15];
      =     "Op10.Bench.Systems".Command.Abbassa_index_cassetto;
      A     "Op10.Cycles".General.State.State_Bit[16];
      A     "Op10.Bench.Systems".State.Cassetto_dentro;
      O(;
      A     "Op10.Cycles".General.State.State_Bit[40];
      O     "Op10.Cycles".Restore.State.State_Bit[20];
      A     "Op10.Bench.Systems".State.Cassetto_fuori;
      );
      =     "Op10.Bench.Systems".Command.Alza_index_cassetto;
//*************************** COMANDI SENZA INTERBLOCCHI ***************
//CMD---------->Comando abbassa index cassetto
//MANUALE
      A     "Line.OperatorPanel".Commands.Man_10_IndexCassetto;
      A     "Line.MapE".Jog_meno;
      A     "OP10".Mode.Manual;
//AUTOMATICO
      O(;
      A     "OP10".Mode.Automatic;
      AN    "OP10".Diagnostic.Hold_State;
      A     "Op10.Bench.Systems".Command.Abbassa_index_cassetto;
      );
//SICUREZZA
      A     "OP10".Diagnostic.Safe_State;
      =     #Cmd_abbassa_indc;
//CMD---------->Comando alza index cassetto
//MANUALE
      A     "Line.OperatorPanel".Commands.Man_10_IndexCassetto;
      A     "Line.MapE".Jog_piu;
      A     "OP10".Mode.Manual;
//AUTOMATICO
      O(;
      A     "OP10".Mode.Automatic;
      AN    "OP10".Diagnostic.Hold_State;
      A     "Op10.Bench.Systems".Command.Alza_index_cassetto;
      );
//SICUREZZA
      A     "OP10".Diagnostic.Safe_State;
      =     #Cmd_alza_indc;
//************************** INTERBLOCCHI (E SEGNALAZIONE) ****************************
      A     "Op10.Bench.Systems".Command.Reset_allarmi;
      O     "Op10.Bench.Systems".State.Cassetto_dentro;
      O     "Op10.Bench.Systems".State.Cassetto_fuori;
      R     "Op10.Bench.Alarms".Warning.Alarm01;
      A     #Cmd_alza_indc;
      A(;
      AN    "Op10.Bench.Systems".State.Cassetto_dentro;
      AN    "Op10.Bench.Systems".State.Cassetto_fuori;
      );
      S     "Op10.Bench.Alarms".Warning.Alarm01;
// MSG sblocco solo con ribaditrice alta
      A     "Op10.Bench.Systems".Command.Reset_allarmi;
      O     "Op10.Bench.Systems".State.Ribaditrice_alta;
      R     "Op10.Bench.Alarms".Warning.Alarm03;
      A     #Cmd_abbassa_indc;
      AN    "Op10.Bench.Systems".State.Ribaditrice_alta;
      S     "Op10.Bench.Alarms".Warning.Alarm03;
// MSG sblocco solo con assi fermi
      A     "Op10.Bench.Systems".Command.Reset_allarmi;
      O     "Op10.Bench.Systems".State.Assi_fermi;
      R     "Op10.Bench.Alarms".Warning.Alarm04;
      A     #Cmd_abbassa_indc;
      AN    "Op10.Bench.Systems".State.Assi_fermi;
      S     "Op10.Bench.Alarms".Warning.Alarm04;
// MSG sblocco solo con pezzo bloccato
      A     "Op10.Bench.Systems".Command.Reset_allarmi;
      O     "Op10.Bench.Systems".State.Pezzo_sbloccato;
      R     "Op10.Bench.Alarms".Warning.Alarm05;
      A     #Cmd_abbassa_indc;
      AN    "Op10.Bench.Systems".State.Pezzo_sbloccato;
      S     "Op10.Bench.Alarms".Warning.Alarm05;
//************************** COMANDI CON INTERBLOCCHI ******************************
      AN    "Op10.Bench.Alarms".Warning.Alarm03;
      AN    "Op10.Bench.Alarms".Warning.Alarm04;
      AN    "Op10.Bench.Alarms".Warning.Alarm05;
      A     #Cmd_abbassa_indc;
      =     #Cmd_abbassa_indc_ibl;
      AN    "Op10.Bench.Alarms".Warning.Alarm01;
      A     #Cmd_alza_indc;
      =     #Cmd_alza_indc_ibl;
      CALL  "Std System.Cylinder" , "Ist_cil_10_Index_cass" (
           IN_Enable                := TRUE,
           IN_Command_CylForward    := #Cmd_alza_indc_ibl,
           IN_Command_CylBack       := #Cmd_abbassa_indc_ibl,
           IN_EndStroke_Forward     := "Op10.Bench.MapE".Index_cassetto_Su,
           IN_EndStroke_Back        := "Op10.Bench.MapE".Index_cassetto_Giu,
           IN_Alarms_Reset          := "Op10.Bench.Systems".Command.Reset_allarmi,
           IN_Alarms_TimeOut        := T#2S,
           IN_Hold_Condition        := FALSE,
           OUT_EV_Forward           := "Op10.Bench.MapA".EV_alza_index_cassetto,
           OUT_EV_Back              := "Op10.Bench.MapA".EV_abb_index_cassetto,
           OUT_State_CylForward     := "Op10.Bench.Systems".State.Index_cassetto_alto,
           OUT_State_CylBack        := "Op10.Bench.Systems".State.Index_cassetto_basso,
           OUT_Alarm_ES_Forward     := "Op10.Bench.Alarms".StopCycle.Alarm03,
           OUT_Alarm_ES_Back        := "Op10.Bench.Alarms".StopCycle.Alarm04,
           OUT_Alarm_ForwBack       := "Op10.Bench.Alarms".StopCycle.Alarm05);
NETWORK
TITLE = Blocco/Sblocco pezzo
//*************************** COMANDI DA CICLI *************************
      A     "Op10.Cycles".General.State.State_Bit[40];
      O     "Op10.Cycles".Restore.State.State_Bit[20];
      A     "Op10.Bench.MapE".Index_cassetto_Su;
      A     "Op10.Bench.Systems".State.Cassetto_fuori;
      =     "Op10.Bench.Systems".Command.Sblocca_pezzo;
      A     "Op10.Cycles".General.State.State_Bit[13];
      O     "Op10.Cycles".General.State.State_Bit[16];
      =     "Op10.Bench.Systems".Command.Blocca_pezzo;
//*************************** COMANDI SENZA INTERBLOCCHI ***************
//CMD---------->Comando sblocco
//MANUALE
      A     "Line.OperatorPanel".Commands.Man_10_BloccoPezzo;
      A     "Line.MapE".Jog_piu;
      A     "OP10".Mode.Manual;
//AUTOMATICO
      O(;
      A     "OP10".Mode.Automatic;
      AN    "OP10".Diagnostic.Hold_State;
      A     "Op10.Bench.Systems".Command.Sblocca_pezzo;
      );
//SICUREZZA
      A     "OP10".Diagnostic.Safe_State;
      =     #Cmd_sblocca_pezzo;
//CMD---------->Comando alza ribaditrice
//MANUALE
      A     "Line.OperatorPanel".Commands.Man_10_BloccoPezzo;
      A     "Line.MapE".Jog_meno;
      A     "OP10".Mode.Manual;
//AUTOMATICO
      O(;
      A     "OP10".Mode.Automatic;
      AN    "OP10".Diagnostic.Hold_State;
      A     "Op10.Bench.Systems".Command.Blocca_pezzo;
      );
//SICUREZZA
      A     "OP10".Diagnostic.Safe_State;
      =     #Cmd_blocca_pezzo;
//************************** INTERBLOCCHI (E SEGNALAZIONE) ****************************
//MSG---> Segnalazione interblocco Movimento ribaditrice non ammesso con motore ribaditrice in marcia
      A     "Op10.Bench.Systems".Command.Reset_allarmi;
      O(;
      A     "Op10.Bench.Systems".State.Cassetto_fuori;
      A     "Op10.Bench.Systems".State.Index_cassetto_alto;
      );
      R     "Op10.Bench.Alarms".Warning.Alarm02;
      A     #Cmd_sblocca_pezzo;
      A(;
      AN    "Op10.Bench.Systems".State.Cassetto_fuori;
      ON    "Op10.Bench.Systems".State.Index_cassetto_alto;
      );
      S     "Op10.Bench.Alarms".Warning.Alarm02;
//************************** COMANDI CON INTERBLOCCHI ******************************
//CMD-------------> Comando abbassa e alza
      AN    "Op10.Bench.Alarms".Warning.Alarm02;
      A     #Cmd_sblocca_pezzo;
      =     #Cmd_sblocca_pezzo_ibl;
      A     #Cmd_blocca_pezzo;
      =     #Cmd_blocca_pezzo_ibl;
      CALL  "Std System.Cylinder" , "Ist_10_CilBloccoPezzo" (
           IN_Enable                := TRUE,
           IN_Command_CylForward    := #Cmd_sblocca_pezzo_ibl,
           IN_Command_CylBack       := #Cmd_blocca_pezzo_ibl,
           IN_EndStroke_Forward     := "Op10.Bench.MapE".Sblocco_pezzo_Su,
           IN_EndStroke_Back        := "Op10.Bench.MapE".Sblocco_pezzo_Giu,
           IN_Alarms_Reset          := "Op10.Bench.Systems".Command.Reset_allarmi,
           IN_Alarms_TimeOut        := T#4S,
           IN_Hold_Condition        := FALSE,
           OUT_EV_Forward           := "Op10.Bench.MapA".EV_sblocco_pezzo,
           OUT_EV_Back              := "Op10.Bench.MapA".EV_blocco_pezzo,
           OUT_State_CylForward     := "Op10.Bench.Systems".State.Pezzo_bloccato,
           OUT_State_CylBack        := "Op10.Bench.Systems".State.Pezzo_sbloccato,
           OUT_Alarm_ES_Forward     := "Op10.Bench.Alarms".StopCycle.Alarm06,
           OUT_Alarm_ES_Back        := "Op10.Bench.Alarms".StopCycle.Alarm07,
           OUT_Alarm_ForwBack       := "Op10.Bench.Alarms".StopCycle.Alarm08);
NETWORK
TITLE = Gestione numero ribaditura in corso
      AN    "Op10.Cycles".General.Command.Activate_Cycle;
      O     "Op10.Cycles".General.State.State_Bit[10];
      O     "Op10.Cycles".General.State.State_Bit[16];
      O     "Op10.Cycles".General.State.State_Bit[40];
      JCN   nAzz;
      L     0;
      T     "Op10.Bench.Systems".Data.Num_punto_in_lavorazione;
nAzz: NOP   0;
      A     "Op10.Cycles".General.State.State_Bit[20];
      FP    "AppoFP_M50.3";
      =     "Op10.Bench.Systems".State.FP_stato_20_generale;
      AN    "Op10.Bench.Systems".State.FP_stato_20_generale;
      JC    nIn;
      L     "Op10.Bench.Systems".Data.Num_punto_in_lavorazione;
      L     1;
      +I;
      T     "Op10.Bench.Systems".Data.Num_punto_in_lavorazione;
nIn:  NOP   0;
NETWORK
TITLE = Valori posizione ribaditura corrente
      L     "Op10.Bench.Systems".Data.Num_punto_in_lavorazione;
      L     0;
      >I;
      JC    Cal;
// Punto inesistente
      L     L#0;
      T     "Op10.Bench.Systems".Data.Pos_comandata_asse_X;
      T     "Op10.Bench.Systems".Data.Pos_comandata_asse_Y;
      T     "Op10.Bench.Systems".Data.Tempo_ribaditura;
      JU    Cen;
Cal:  NOP   0;	// Estrazione dati punto da ricetta
      L     "Op10.Bench.Systems".Data.Num_punto_in_lavorazione;
      L     1;
      -I;
      ITD;
      L     L#12;
      *D;
      L     L#82;
      +D;
      SLW   3;
      T     #Punt1;
      OPN   "Op10.Bench.Recipe";
      L     DBD [#Punt1];
      T     #Pos_comandata_asse_X;
      L     #Punt1;
      L     32;
      +D;
      T     #Punt1;
      L     DBD [#Punt1];
      T     #Pos_comandata_asse_Y;
      L     #Punt1;
      L     32;
      +D;
      T     #Punt1;
      L     DBD [#Punt1];
      T     #Tempo_ribaditura;
      L     #Pos_comandata_asse_X;
      T     "Op10.Bench.Systems".Data.Pos_comandata_asse_X;
      L     #Pos_comandata_asse_Y;
      T     "Op10.Bench.Systems".Data.Pos_comandata_asse_Y;
      L     #Tempo_ribaditura;
      T     "Op10.Bench.Systems".Data.Tempo_ribaditura;
Cen:  NOP   0;
NETWORK
TITLE = Impegno, comandi e stati ribaditrice per lavoro su OP10
      A     "Op10.Cycles".General.State.State_Bit[16];
      O     "Op10.Cycles".General.State.State_Bit[20];
      O     "Op10.Cycles".General.State.State_Bit[25];
      O     "Op10.Cycles".General.State.State_Bit[30];
      A     "Op10.Cycles".General.Command.Activate_Cycle;
      O(;
      A     "Op10.Cycles".Restore.State.State_Bit[10];
      A     "Op10.Cycles".Restore.Command.Activate_Cycle;
      );
      =     "Op10.Bench.Systems".Command.Prenota_ribaditrice;
      A     "Op10.Cycles".General.State.State_Bit[20];
      O     "Op10.Cycles".General.State.State_Bit[25];
      O     "Op10.Cycles".General.State.State_Bit[30];
      =     "Op10.Bench.Systems".Command.Marcia_ribaditrice;
      A     "Op10.Cycles".General.State.State_Bit[25];
      A     "Op10.Bench.Systems".State._Ribaditrice_a_disposiz;
      =     "Op10.Bench.Systems".Command.Abbassa_ribaditrice;
      A     "Op10.Cycles".General.State.State_Bit[13];
      AN    "Op10.Bench.Systems".State._Ribad_in_fuori_ingombro;
      O     "Op10.Cycles".General.State.State_Bit[30];
      O     "Op10.Cycles".Restore.State.State_Bit[10];
      A     "Op10.Bench.Systems".State._Ribaditrice_a_disposiz;
      =     "Op10.Bench.Systems".Command.Alza_ribaditrice;
      A     "Line.Systems".State.Ribad_prenotata_da_OP10;
      =     "Op10.Bench.Systems".State._Ribaditrice_a_disposiz;
NETWORK
TITLE = Ribaditura
      L     "Op10.Bench.Systems".Data.Tempo_ribaditura;
      T     #TempoTime;
      CALL  "TIM_S5TI" (
           $1                       := #TempoTime,
           $2                       := #TempoS5T);
      A     "Op10.Cycles".General.State.State_Bit[25];
      A     "Op10.Bench.Systems".State.Ribaditrice_in_marcia;
      A     "Op10.Bench.Systems".State.Ribaditrice_bassa;
      L     #TempoS5T;
      SD    "Op10_Tempo_di_ribaditura";
      A     "Op10_Tempo_di_ribaditura";
      =     "Op10.Bench.Systems".State.Ribaditura_effettuata;
NETWORK
TITLE = Assi - movimenti per lavorazioni OP10
      A     "Op10.Cycles".General.State.State_Bit[20];
      A     "Line.Systems".State.Ribad_prenotata_da_OP10;
      =     "Op10.Bench.Systems".Command.Vai_in_posizione_assi;
      A     "Line.Systems".State.AsseX_posizioneRaggiunta;
      A     "Line.Systems".State.AsseY_posizioneRaggiunta;
      A     "Line.Systems".State.Ribad_prenotata_da_OP10;
      =     "Op10.Bench.Systems".State._Assi_posiz_raggiunta;
NETWORK
TITLE = Definizione pezzo buono o scarto
      A     "Op10.Cycles".General.State.State_Bit[35];
      S     "Op10.Bench.Systems".State.Ribaditura_pezzo_OK;
      A     "Op10.Bench.MapE".Sblocco_pezzo_Su;
      R     "Op10.Bench.Systems".State.Ribaditura_pezzo_OK;
      A     "Op10.Cycles".Restore.Command.Activate_Cycle;
      A     "Op10.Tools.MapE".Presenza_nozzle_ring;
      AN    "Op10.Bench.Systems".State.Ribaditura_pezzo_OK;
      S     "Op10.Bench.Systems".State.Ribaditura_pezzo_KO;
      A     "Op10.Bench.MapE".Sblocco_pezzo_Su;
      R     "Op10.Bench.Systems".State.Ribaditura_pezzo_KO;
END_FUNCTION

FUNCTION "Op10.Tool.FCMap.E" : VOID	// FC 106
VERSION : 0.1
VAR_INPUT
  ToolType : INT ;
END_VAR
VAR_OUTPUT
  ErrorToolType : BOOL ;
END_VAR
BEGIN
NETWORK
TITLE = Tool 1 - mappa ingressi
// Definizione ingressi E3.0 - E4.6
      L     #ToolType;
      L     1;
      <>I;
      JC    no1;
      SET;
      R     #ErrorToolType;
// Tool 1 - mappa ingressi
      A     I 4.1;
      =     "Op10.Tools.MapE".ToolCode_Bit_0;
      A     I 4.2;
      =     "Op10.Tools.MapE".ToolCode_Bit_1;
      A     I 4.3;
      =     "Op10.Tools.MapE".ToolCode_Bit_2;
      A     I 4.4;
      =     "Op10.Tools.MapE".ToolCode_Bit_3;
      A     I 4.5;
      =     "Op10.Tools.MapE".ToolCode_Bit_4;
      A     I 4.0;
      =     "Op10.Tools.MapE".Anello_1_Inserito;
      A     I 3.7;
      =     "Op10.Tools.MapE".Anello_2_Inserito;
      A     I 3.6;
      =     "Op10.Tools.MapE".Presenza_nozzle_ring;
      A     I 3.1;
      =     "Op10.Tools.MapE".Spacer_1_presente;
      A     I 3.0;
      =     "Op10.Tools.MapE".Spacer_1_invertito;
      A     I 3.3;
      =     "Op10.Tools.MapE".Spacer_2_presente;
      A     I 3.2;
      =     "Op10.Tools.MapE".Spacer_2_invertito;
      A     I 3.5;
      =     "Op10.Tools.MapE".Spacer_3_presente;
      A     I 3.4;
      =     "Op10.Tools.MapE".Spacer_3_invertito;
      BEU;
no1:  NOP   0;
NETWORK
TITLE = Tool 2 - mappa ingressi
      L     #ToolType;
      L     2;
      <>I;
      JC    no2;
      SET;
      S     #ErrorToolType;
// Tool 2 - predisposto ma inesistente
      BEU;
no2:  NOP   0;
NETWORK
TITLE = Error Tool Type
      SET;
      S     #ErrorToolType;
END_FUNCTION

FUNCTION "Op10.FCCycles" : VOID	// FC 120
VERSION : 0.1
BEGIN
NETWORK
TITLE =
      A     "OP10".Mode.Automatic;
      FP    "AppoFP_M50.4";
      =     "Op10.Bench.Systems".State.FP_Mode_automatic;
      AN    "OP10".Diagnostic.Alarm_Stop_Cycle;
      AN    "OP10".Diagnostic.Alarm_Emergency;
      FP    "AppoFP_M50.5";
      =     "Op10.Bench.Systems".State.FP_uscita_da_allarme;
NETWORK
TITLE =
      A     "Op10.Bench.Systems".State.FP_Mode_automatic;
      O     "Op10.Bench.Systems".State.FP_uscita_da_allarme;
      A(;
      AN    "Op10.Bench.Systems".State.Cassetto_fuori;
      ON    "Op10.Bench.MapE".Index_cassetto_Su;
      ON    "Op10.Bench.MapE".Sblocco_pezzo_Su;
      );
      S     "Op10.Cycles".Restore.Command.Activate_Cycle;
      AN    "OP10".Mode.Automatic;
//      U     "OP10".Diagnostic.Alarm_Stop_Cycle
      O     "OP10".Diagnostic.Alarm_Emergency;
      O     "Op10.Bench.MapE".PulStopCiclo;
      O     "Op10.Cycles".Restore.State.State_Bit[60];
      R     "Op10.Cycles".Restore.Command.Activate_Cycle;
      CLR;
      =     "OP10".Diagnostic.Hold_State;
      CALL  "Op10.Cycle.Restore" , "Op10.Ist.Cycle.Restore" (
           IN_Cm_ON                 := "Op10.Cycles".Restore.Command.Activate_Cycle,
           IN_HOLD                  := "OP10".Diagnostic.Hold_State,
           IN_STEP                  := FALSE,
           OUT_St_CicloInCorso      := "Op10.Cycles".Restore.State.Cycle_In_Progress,
           OUT_St_CicloTerminatoOK  := "Op10.Cycles".Restore.State.Cycle_Ended_OK,
           OUT_St_CicloTerminatoKO  := "Op10.Cycles".Restore.State.Cycle_Ended_KO,
           OUT_CicloStato           := "Op10.Cycles".Restore.State.State,
           OUT_Page                 := "Op10.Cycles".Restore.State.Page,
           OUT_Message              := "Op10.Cycles".Restore.State.Message);
NETWORK
TITLE =
      A     "OP10".Mode.Automatic;
      AN    "OP10".Diagnostic.Alarm_Stop_Cycle;
      AN    "OP10".Diagnostic.Alarm_Emergency;
      AN    "Op10.Cycles".Restore.Command.Activate_Cycle;
// condizione di sicurezza
      AN    "Op10.Bench.MapE".PulStopCiclo;
      =     "Op10.Cycles".General.Command.Activate_Cycle;
      CALL  "Op10.Cycle.General" , "Op10.Ist.Cycle.General" (
           IN_Cm_ON                 := "Op10.Cycles".General.Command.Activate_Cycle,
           IN_HOLD                  := "OP10".Diagnostic.Hold_State,
           IN_STEP                  := FALSE,
           OUT_St_CicloInCorso      := "Op10.Cycles".General.State.Cycle_In_Progress,
           OUT_St_CicloTerminatoOK  := "Op10.Cycles".General.State.Cycle_Ended_OK,
           OUT_St_CicloTerminatoKO  := "Op10.Cycles".General.State.Cycle_Ended_KO,
           OUT_CicloStato           := "Op10.Cycles".General.State.State,
           OUT_Page                 := "Op10.Cycles".General.State.Page,
           OUT_Message              := "Op10.Cycles".General.State.Message);
END_FUNCTION

FUNCTION "OP20.FCMain" : VOID	// FC 150
VERSION : 0.1
VAR_TEMP
  ErrorToolType : BOOL ;
END_VAR
BEGIN
NETWORK
TITLE =
NETWORK
TITLE = OP20 ToolType error
      CALL  "Op20.Bench.FCMapE";
      CALL  "Op20.Tool.FCMapE" (
           ToolType                 := "Op20.Bench.Recipe".ToolType,
           ErrorToolType            := #ErrorToolType);
      A     #ErrorToolType;
      AN    "Op20.Bench.Recipe".Disable.CkCodicePortapezzo;
      S     "Op20.Bench.Alarms".StopCycle.Alarm07;
      CALL  "Op20.Bench.FCConfig";
NETWORK
TITLE =
      A     "Line.Systems".Command.Reset_allarmi;
      =     "Op20.Bench.Systems".Command.Reset_allarmi;
      A     "Line.Systems".Command.TestLampade;
      =     "Op20.Bench.Systems".Command.TestLampade;
      A     "Line.Systems".State.Porte_chiuse;
      =     "Op20.Bench.Systems".State.Porte_chiuse;
      A     "Line.Systems".State.Porte_chiuse_e_bloccate;
      =     "Op20.Bench.Systems".State.Porte_chiuse_e_bloccate;
      CALL  "Bench.Alarms" (
           NumDBallarmi             := "Op20.Bench.Alarms",
           Reset_Allarmi            := "Op20.Bench.Systems".Command.Reset_allarmi,
           AllarmeEmergenza         := "OP20".Diagnostic.Alarm_Emergency,
           AllarmeStopCiclo         := "OP20".Diagnostic.Alarm_Stop_Cycle,
           AllarmeStartCiclo        := "OP20".Diagnostic.Alarm_No_Restart,
           AllarmeWarning           := "OP20".Diagnostic.Alarm_Warning);
// Bench mode = Line mode...
      A     "Line".Mode.Emergency;
      =     "OP20".Mode.Emergency;
      A     "Line".Mode.Test_Machine;
      =     "OP20".Mode.Test_Machine;
      A     "Line".Mode.Setup;
      =     "OP20".Mode.Setup;
      A     "Line".Mode.Manual;
      =     "OP20".Mode.Manual;
      A     "Line".Mode.Automatic;
      =     "OP20".Mode.Automatic;
NETWORK
TITLE =
      CALL  "Op20.Bench.FCSystems";
      CALL  "Op20.FCCycles";
NETWORK
TITLE =
      CALL  "Op20.Bench.FCMapA";
END_FUNCTION

FUNCTION "Op20.Bench.FCMapE" : VOID	// FC 151
VERSION : 0.1
VAR_TEMP
  RetVal : WORD ;
  Tastatore : REAL ;
END_VAR
BEGIN
NETWORK
TITLE =
      A     I 10.4;
      =     "Op20.Bench.MapE".Cassetto_dentro;
      A     I 10.6;
      =     "Op20.Bench.MapE".Index_cassetto_Giu;
      A     I 10.5;
      =     "Op20.Bench.MapE".Index_cassetto_Su;
      A     I 10.3;
      =     "Op20.Bench.MapE".Piantaggio_Giu;
      A     I 10.2;
      =     "Op20.Bench.MapE".Piantaggio_Su;
      A     I 10.1;
      =     "Op20.Bench.MapE".Gruppo_piantaggio_Giu;
      A     I 10.0;
      =     "Op20.Bench.MapE".Gruppo_piantaggio_Su;
NETWORK
TITLE =
      CALL  "SCALE" (
           $1                       := P#P 256.0,
           $2                       := L#1088421888,
           $3                       := L#0,
           $4                       := FALSE,
           $5                       := #RetVal,
           $6                       := #Tastatore);
      L     #Tastatore;
      L     "Op20.Bench.Config".Offset_Tastatore;
      -R;
      T     "Op20.Bench.MapE"._Posizione_Punzone;
END_FUNCTION

FUNCTION "Op20.Bench.FCMapA" : VOID	// FC 152
VERSION : 0.1
BEGIN
NETWORK
TITLE =
      A     "Op20.Bench.MapA".Fine_ciclo_OK;
      =     Q 0.5;
      A     "Op20.Bench.MapA".Fine_ciclo_NON_OK;
      =     Q 0.6;
      A     "Op20.Bench.MapA".EV_abb_index_cassetto;
      =     Q 2.0;
      A     "Op20.Bench.MapA".EV_alza_index_cassetto;
      =     Q 2.1;
      A     "Op20.Bench.MapA".EV_abbassa_piantaggio;
      =     Q 1.5;
      A     "Op20.Bench.MapA".EV_alza_piantaggio;
      =     Q 1.6;
      A     "Op20.Bench.MapA".EV_abb_grupp_piantaggio;
      =     Q 1.3;
      A     "Op20.Bench.MapA".EV_alz_grupp_piantaggio;
      =     Q 1.4;
END_FUNCTION

FUNCTION "Op20.Bench.FCConfig" : VOID	// FC 153
VERSION : 0.1
BEGIN
NETWORK
TITLE =
// Impostato da pagina di configurazione su PO
//      L     3.808000e+000
//      T     "Op20.Bench.Config".Offset_Tastatore
END_FUNCTION

FUNCTION "Op20.Bench.FCSystems" : VOID	// FC 155
VERSION : 0.1
VAR_TEMP
  Cmd_abbassa_indc : BOOL ;
  Cmd_alza_indc : BOOL ;
  Cmd_abbassa_indc_ibl : BOOL ;
  Cmd_alza_indc_ibl : BOOL ;
  Cmd_sblocca_pezzo : BOOL ;
  Cmd_blocca_pezzo : BOOL ;
  Cmd_sblocca_pezzo_ibl : BOOL ;
  Cmd_blocca_pezzo_ibl : BOOL ;
  Cmd_AlzaGrPiant : BOOL ;
  Cmd_AbbassaGrPiant : BOOL ;
  Cmd_AlzaGrPiant_ibl : BOOL ;
  Cmd_AbbassaGrPiant_ibl : BOOL ;
  Cmd_AlzaPiant : BOOL ;
  Cmd_AbbassaPiant : BOOL ;
  Cmd_AlzaPiant_ibl : BOOL ;
  Cmd_AbbassaPiant_ibl : BOOL ;
  CorsaMinRaggiunta : BOOL ;
  CorsaMaxSuperata : BOOL ;
  TempoTime : TIME ;
  TempoS5T : S5TIME ;
END_VAR
BEGIN
NETWORK
TITLE = ******************       Diagnostica       *******************
NETWORK
TITLE = Allarmi di emergenza
NETWORK
TITLE = Controllo toolcode 
      L     DB156.DBB 0;
      L     W#16#1F;
      AW;
      L     DB160.DBW 24;
      <>I;
      A     "Op20.Bench.Recipe".Disable.CkCodicePortapezzo;
      S     "Op20.Bench.Alarms".StopCycle.Alarm08;
NETWORK
TITLE = Allarmi di STOP CICLO
NETWORK
TITLE = Allarmi di NON START CICLO
NETWORK
TITLE = Allarmi di Warning
NETWORK
TITLE = Diagnostica: Hold Macchina
      AN    "OP20".Diagnostic.Alarm_Emergency;
      A(;
      A     "OP20".Mode.Automatic;
      AN    "OP20".Diagnostic.Alarm_Stop_Cycle;
      A     "Op20.Bench.Systems".State.Porte_chiuse_e_bloccate;
      O(;
      A     "OP20".Mode.Manual;
      A     "Op20.Bench.Systems".State.Porte_chiuse;
      );
      );
      =     "OP20".Diagnostic.Safe_State;
NETWORK
TITLE = ******************          Stati            *******************
      AN    "Op20.Bench.MapE".Cassetto_dentro;
      =     "Op20.Bench.Systems".State.Cassetto_fuori;
      A     "Op20.Bench.MapE".Cassetto_dentro;
      =     "Op20.Bench.Systems".State.Cassetto_dentro;
NETWORK
TITLE = Stato: Fronte Start Ciclo
NETWORK
TITLE = Lampade
      A     "Op20.Bench.Systems".State.Piantaggio_pezzo_OK;
      A     "OP20".Mode.Automatic;
      O     "Op20.Bench.Systems".Command.TestLampade;
      =     "Op20.Bench.MapA".Fine_ciclo_OK;
      A     "Op20.Bench.Systems".State.Piantaggio_pezzo_KO;
      A     "OP20".Mode.Automatic;
      O     "Op20.Bench.Systems".Command.TestLampade;
      =     "Op20.Bench.MapA".Fine_ciclo_NON_OK;
NETWORK
TITLE = Cycle Type
NETWORK
TITLE = ******************         Sistemi           *******************
NETWORK
TITLE = Alza/abbassa Index cassetto
//*************************** COMANDI DA CICLI *************************
      A     "Op20.Cycles".General.State.State_Bit[35];
      O     "Op20.Cycles".Restore.State.State_Bit[15];
      =     "Op20.Bench.Systems".Command.Abbassa_index_cassetto;
      A     "Op20.Cycles".General.State.State_Bit[15];
      =     "Op20.Bench.Systems".Command.Alza_index_cassetto;
//*************************** COMANDI SENZA INTERBLOCCHI ***************
//CMD---------->Comando abbassa index cassetto
//MANUALE
      A     "Line.OperatorPanel".Commands.Man_20_IndexCassetto;
      A     "Line.MapE".Jog_meno;
      A     "OP20".Mode.Manual;
//AUTOMATICO
      O(;
      A     "OP20".Mode.Automatic;
      AN    "OP20".Diagnostic.Hold_State;
      A     "Op20.Bench.Systems".Command.Abbassa_index_cassetto;
      );
//SICUREZZA
      A     "OP20".Diagnostic.Safe_State;
      =     #Cmd_abbassa_indc;
//CMD---------->Comando alza index cassetto
//MANUALE
      A     "Line.OperatorPanel".Commands.Man_20_IndexCassetto;
      A     "Line.MapE".Jog_piu;
      A     "OP20".Mode.Manual;
//AUTOMATICO
      O(;
      A     "OP20".Mode.Automatic;
      AN    "OP20".Diagnostic.Hold_State;
      A     "Op20.Bench.Systems".Command.Alza_index_cassetto;
      );
//SICUREZZA
      A     "OP20".Diagnostic.Safe_State;
      =     #Cmd_alza_indc;
//************************** INTERBLOCCHI (E SEGNALAZIONE) ****************************
      A     "Op20.Bench.Systems".Command.Reset_allarmi;
      O     "Op20.Bench.Systems".State.Cassetto_dentro;
      O     "Op20.Bench.Systems".State.Cassetto_fuori;
      R     "Op20.Bench.Alarms".Warning.Alarm01;
      A     #Cmd_alza_indc;
      AN    "Op20.Bench.Systems".State.Cassetto_dentro;
      S     "Op20.Bench.Alarms".Warning.Alarm01;
// Msg 
      A     "Op20.Bench.Systems".Command.Reset_allarmi;
      O(;
      A     "Op20.Bench.Systems".State.Gruppo_piantaggio_alto;
      A     "Op20.Bench.Systems".State.Piantaggio_alto;
      );
      R     "Op20.Bench.Alarms".Warning.Alarm05;
      AN    "Op20.Bench.Systems".State.Gruppo_piantaggio_alto;
      ON    "Op20.Bench.Systems".State.Piantaggio_alto;
      A     #Cmd_abbassa_indc;
      S     "Op20.Bench.Alarms".Warning.Alarm05;
//************************** COMANDI CON INTERBLOCCHI ******************************
      AN    "Op20.Bench.Alarms".Warning.Alarm05;
      A     #Cmd_abbassa_indc;
      =     #Cmd_abbassa_indc_ibl;
      AN    "Op20.Bench.Alarms".Warning.Alarm01;
      A     #Cmd_alza_indc;
      =     #Cmd_alza_indc_ibl;
      CALL  "Std System.Cylinder" , "Ist_cil_20_Index_cass" (
           IN_Enable                := TRUE,
           IN_Command_CylForward    := #Cmd_alza_indc_ibl,
           IN_Command_CylBack       := #Cmd_abbassa_indc_ibl,
           IN_EndStroke_Forward     := "Op20.Bench.MapE".Index_cassetto_Su,
           IN_EndStroke_Back        := "Op20.Bench.MapE".Index_cassetto_Giu,
           IN_Alarms_Reset          := "Op20.Bench.Systems".Command.Reset_allarmi,
           IN_Alarms_TimeOut        := T#1S500MS,
           IN_Hold_Condition        := FALSE,
           OUT_EV_Forward           := "Op20.Bench.MapA".EV_alza_index_cassetto,
           OUT_EV_Back              := "Op20.Bench.MapA".EV_abb_index_cassetto,
           OUT_State_CylForward     := "Op20.Bench.Systems".State.Index_cassetto_alto,
           OUT_State_CylBack        := "Op20.Bench.Systems".State.Index_cassetto_basso,
           OUT_Alarm_ES_Forward     := "Op20.Bench.Alarms".StopCycle.Alarm02,
           OUT_Alarm_ES_Back        := "Op20.Bench.Alarms".StopCycle.Alarm03,
           OUT_Alarm_ForwBack       := "Op20.Bench.Alarms".StopCycle.Alarm04);
NETWORK
TITLE = Alza/abbassa gruppo di piantaggio
//*************************** COMANDI DA CICLI *************************
      A     "Op20.Cycles".General.State.State_Bit[30];
      O     "Op20.Cycles".Restore.State.State_Bit[10];
      A     "Op20.Bench.Systems".State.Piantaggio_alto;
      =     "Op20.Bench.Systems".Command.Alza_gruppo_piantaggio;
      A     "Op20.Cycles".General.State.State_Bit[20];
      =     "Op20.Bench.Systems".Command.Abbasa_gruppo_piantaggio;
//*************************** COMANDI SENZA INTERBLOCCHI ***************
//CMD---------->Comando alza gruppo
//MANUALE
      A     "Line.OperatorPanel".Commands.Man_20_GruppoPiantaggio;
      A     "Line.MapE".Jog_meno;
      A     "OP20".Mode.Manual;
//AUTOMATICO
      O(;
      A     "OP20".Mode.Automatic;
      AN    "OP20".Diagnostic.Hold_State;
      A     "Op20.Bench.Systems".Command.Alza_gruppo_piantaggio;
      );
//SICUREZZA
//      U     "OP20".Diagnostic.Safe_State
      A     "Op20.Bench.Systems".State.Porte_chiuse;
      =     #Cmd_AlzaGrPiant;
//CMD---------->Comando abbassa gruppo
//MANUALE
      A     "Line.OperatorPanel".Commands.Man_20_GruppoPiantaggio;
      A     "Line.MapE".Jog_piu;
      A     "OP20".Mode.Manual;
//AUTOMATICO
      O(;
      A     "OP20".Mode.Automatic;
      AN    "OP20".Diagnostic.Hold_State;
      A     "Op20.Bench.Systems".Command.Abbasa_gruppo_piantaggio;
      );
//SICUREZZA
      A     "OP20".Diagnostic.Safe_State;
      =     #Cmd_AbbassaGrPiant;
//************************** INTERBLOCCHI (E SEGNALAZIONE) ****************************
      A     "Op20.Bench.Systems".Command.Reset_allarmi;
      O     "Op20.Bench.Systems".State.Cassetto_dentro;
      R     "Op20.Bench.Alarms".Warning.Alarm06;
      A     #Cmd_AbbassaGrPiant;
      AN    "Op20.Bench.Systems".State.Cassetto_dentro;
      S     "Op20.Bench.Alarms".Warning.Alarm06;
      A     "Op20.Bench.Systems".Command.Reset_allarmi;
      O     "Op20.Bench.Systems".State.Index_cassetto_alto;
      R     "Op20.Bench.Alarms".Warning.Alarm07;
      A     #Cmd_AbbassaGrPiant;
      AN    "Op20.Bench.Systems".State.Index_cassetto_alto;
      S     "Op20.Bench.Alarms".Warning.Alarm07;
      A     "Op20.Bench.Systems".Command.Reset_allarmi;
      O     "Op20.Bench.Systems".State.Piantaggio_alto;
      R     "Op20.Bench.Alarms".Warning.Alarm09;
      A     #Cmd_AlzaGrPiant;
      AN    "Op20.Bench.Systems".State.Piantaggio_alto;
      S     "Op20.Bench.Alarms".Warning.Alarm09;
//************************** COMANDI CON INTERBLOCCHI ******************************
      AN    "Op20.Bench.Alarms".Warning.Alarm09;
      A     #Cmd_AlzaGrPiant;
      =     #Cmd_AlzaGrPiant_ibl;
      AN    "Op20.Bench.Alarms".Warning.Alarm06;
      AN    "Op20.Bench.Alarms".Warning.Alarm07;
      A     #Cmd_AbbassaGrPiant;
      =     #Cmd_AbbassaGrPiant_ibl;
      CALL  "Std System.Cylinder" , "Ist_cil_20_gr_piantaggio" (
           IN_Enable                := TRUE,
           IN_Command_CylForward    := #Cmd_AbbassaGrPiant_ibl,
           IN_Command_CylBack       := #Cmd_AlzaGrPiant_ibl,
           IN_EndStroke_Forward     := "Op20.Bench.MapE".Gruppo_piantaggio_Giu,
           IN_EndStroke_Back        := "Op20.Bench.MapE".Gruppo_piantaggio_Su,
           IN_Alarms_Reset          := "Op20.Bench.Systems".Command.Reset_allarmi,
           IN_Alarms_TimeOut        := T#3S,
           IN_Hold_Condition        := FALSE,
           OUT_EV_Forward           := "Op20.Bench.MapA".EV_abb_grupp_piantaggio,
           OUT_EV_Back              := "Op20.Bench.MapA".EV_alz_grupp_piantaggio,
           OUT_State_CylForward     := "Op20.Bench.Systems".State.Gruppo_piantaggio_basso,
           OUT_State_CylBack        := "Op20.Bench.Systems".State.Gruppo_piantaggio_alto,
           OUT_Alarm_ES_Forward     := "Op20.Bench.Alarms".StopCycle.Alarm01,
           OUT_Alarm_ES_Back        := "Op20.Bench.Alarms".StopCycle.Alarm02,
           OUT_Alarm_ForwBack       := "Op20.Bench.Alarms".StopCycle.Alarm03);
NETWORK
TITLE = Alza/abbassa cilindro di piantaggio
//*************************** COMANDI DA CICLI *************************
      A     "Op20.Cycles".General.State.State_Bit[30];
      O     "Op20.Cycles".Restore.State.State_Bit[10];
      =     "Op20.Bench.Systems".Command.Alza_piantaggio;
      A     "Op20.Cycles".General.State.State_Bit[25];
      =     "Op20.Bench.Systems".Command.Abbasa_piantaggio;
//*************************** COMANDI SENZA INTERBLOCCHI ***************
//CMD---------->Comando alza gruppo
//MANUALE
      A     "Line.OperatorPanel".Commands.Man_20_Piantaggio;
      A     "Line.MapE".Jog_meno;
      A     "OP20".Mode.Manual;
//AUTOMATICO
      O(;
      A     "OP20".Mode.Automatic;
      AN    "OP20".Diagnostic.Hold_State;
      A     "Op20.Bench.Systems".Command.Alza_piantaggio;
      );
//SICUREZZA
      A     "OP20".Diagnostic.Safe_State;
      =     #Cmd_AlzaPiant;
//CMD---------->Comando abbassa gruppo
//MANUALE
      A     "Line.OperatorPanel".Commands.Man_20_Piantaggio;
      A     "Line.MapE".Jog_piu;
      A     "OP20".Mode.Manual;
//AUTOMATICO
      O(;
      A     "OP20".Mode.Automatic;
      AN    "OP20".Diagnostic.Hold_State;
      A     "Op20.Bench.Systems".Command.Abbasa_piantaggio;
      );
//SICUREZZA
      A     "OP20".Diagnostic.Safe_State;
      =     #Cmd_AbbassaPiant;
//************************** INTERBLOCCHI (E SEGNALAZIONE) ****************************
      A     #Cmd_AbbassaPiant;
      AN    "Op20.Bench.Systems".State.Cassetto_dentro;
      S     "Op20.Bench.Alarms".Warning.Alarm06;
      A     #Cmd_AbbassaPiant;
      AN    "Op20.Bench.Systems".State.Index_cassetto_alto;
      S     "Op20.Bench.Alarms".Warning.Alarm07;
      A     "Op20.Bench.Systems".Command.Reset_allarmi;
      O     "Op20.Bench.Systems".State.Gruppo_piantaggio_basso;
      R     "Op20.Bench.Alarms".Warning.Alarm08;
      A     #Cmd_AbbassaPiant;
      AN    "Op20.Bench.Systems".State.Gruppo_piantaggio_basso;
      S     "Op20.Bench.Alarms".Warning.Alarm08;
//************************** COMANDI CON INTERBLOCCHI ******************************
      A     #Cmd_AlzaPiant;
      =     #Cmd_AlzaPiant_ibl;
      AN    "Op20.Bench.Alarms".Warning.Alarm06;
      AN    "Op20.Bench.Alarms".Warning.Alarm07;
      AN    "Op20.Bench.Alarms".Warning.Alarm08;
      A     #Cmd_AbbassaPiant;
      =     #Cmd_AbbassaPiant_ibl;
      CALL  "Std System.Cylinder" , "Ist_cil_20_piantaggio" (
           IN_Enable                := TRUE,
           IN_Command_CylForward    := #Cmd_AbbassaPiant_ibl,
           IN_Command_CylBack       := #Cmd_AlzaPiant_ibl,
           IN_EndStroke_Forward     := "Op20.Bench.MapE".Piantaggio_Giu,
           IN_EndStroke_Back        := "Op20.Bench.MapE".Piantaggio_Su,
           IN_Alarms_Reset          := "Op20.Bench.Systems".Command.Reset_allarmi,
           IN_Alarms_TimeOut        := T#10S,
           IN_Hold_Condition        := FALSE,
           OUT_EV_Forward           := "Op20.Bench.MapA".EV_abbassa_piantaggio,
           OUT_EV_Back              := "Op20.Bench.MapA".EV_alza_piantaggio,
           OUT_State_CylForward     := "Op20.Bench.Systems".State.Piantaggio_basso,
           OUT_State_CylBack        := "Op20.Bench.Systems".State.Piantaggio_alto,
           OUT_Alarm_ES_Forward     := "Op20.Bench.Alarms".StopCycle.Alarm04,
           OUT_Alarm_ES_Back        := "Op20.Bench.Alarms".StopCycle.Alarm05,
           OUT_Alarm_ForwBack       := "Op20.Bench.Alarms".StopCycle.Alarm06);
NETWORK
TITLE = Pressatua: controllo ciclo e definizione pezzo OK/KO
      L     "Op20.Bench.MapE"._Posizione_Punzone;
      L     "Op20.Bench.Recipe".Corsa_piantaggio_min;
      >=R;
      =     #CorsaMinRaggiunta;
      L     "Op20.Bench.MapE"._Posizione_Punzone;
      L     "Op20.Bench.Recipe".Corsa_piantaggio_max;
      >=R;
      =     #CorsaMaxSuperata;
// gestione timeout piantaggio
      L     "Op20.Bench.Recipe".Timeout_piantaggio;
      T     #TempoTime;
      CALL  "TIM_S5TI" (
           $1                       := #TempoTime,
           $2                       := #TempoS5T);
      A     "Op20.Cycles".General.State.State_Bit[25];
      L     #TempoS5T;
      SD    "OP20_TimeoutPiantaggio";
// Tempo di piantagio
      L     "Op20.Bench.Recipe".Tempo_stabilizzazione;
      T     #TempoTime;
      CALL  "TIM_S5TI" (
           $1                       := #TempoTime,
           $2                       := #TempoS5T);
      A     "Op20.Cycles".General.State.State_Bit[25];
      A     #CorsaMinRaggiunta;
      L     #TempoS5T;
      SD    "OP20_TempoDiPiantaggio";
// definizione pezzo buono o scartgo
      A     "OP20_TimeoutPiantaggio";
      O     #CorsaMaxSuperata;
      A     "Op20.Cycles".General.State.State_Bit[25];
      O     "Op20.Cycles".Restore.Command.Activate_Cycle;
      S     "Op20.Bench.Systems".State.Piantaggio_pezzo_KO;
      A     "OP20_TempoDiPiantaggio";
      A     "Op20.Cycles".General.State.State_Bit[25];
      S     "Op20.Bench.Systems".State.Piantaggio_pezzo_OK;
      A     "Op20.Cycles".General.State.State_Bit[15];
      R     "Op20.Bench.Systems".State.Piantaggio_pezzo_KO;
      R     "Op20.Bench.Systems".State.Piantaggio_pezzo_OK;
// fine operazione di piantaggio
      A     "OP20_TempoDiPiantaggio";
      O     "OP20_TimeoutPiantaggio";
      A     "Op20.Cycles".General.State.State_Bit[25];
      =     "Op20.Bench.Systems".State.Piantaggiofinito;
END_FUNCTION

FUNCTION "Op20.Tool.FCMapE" : VOID	// FC 156
VERSION : 0.1
VAR_INPUT
  ToolType : INT ;
END_VAR
VAR_OUTPUT
  ErrorToolType : BOOL ;
END_VAR
BEGIN
NETWORK
TITLE = Tool 1 - mappa ingressi
      L     #ToolType;
      L     1;
      <>I;
      JC    no1;
      SET;
      R     #ErrorToolType;
// Tool 1 - mappa ingressi
      A     I 2.3;
      =     "Op20.Tools.MapE".ToolCode_Bit_0;
      A     I 2.4;
      =     "Op20.Tools.MapE".ToolCode_Bit_1;
      A     I 2.5;
      =     "Op20.Tools.MapE".ToolCode_Bit_2;
      A     I 2.6;
      =     "Op20.Tools.MapE".ToolCode_Bit_3;
      A     I 2.7;
      =     "Op20.Tools.MapE".ToolCode_Bit_4;
      BEU;
no1:  NOP   0;
NETWORK
TITLE = Tool 2 - mappa ingressi
      L     #ToolType;
      L     2;
      <>I;
      JC    no2;
      SET;
      S     #ErrorToolType;
// Tool 2 - predisposto ma inesistente
      BEU;
no2:  NOP   0;
NETWORK
TITLE = Error Tool Type
      SET;
      S     #ErrorToolType;
END_FUNCTION

